		IF NOT DilSendCmd.bBusy THEN
			IF DilSendCmd.bError THEN
				bError := TRUE;
				nErrorId := DilSendCmd.nErrorId;
				bBusy:= FALSE;
			ELSE
				nState := 4;
			END_IF
			DilSendCmd(bExecute:= FALSE);
		ELSE
			RETURN;
		END_IF
	ELSIF nState = 4 THEN	//Ausgangsposition DilSrc erreicht?
		fbGetPlungerPos(bExecute:= TRUE, DilSendCmd:= DilSendCmd, pDilRef:= pDilRefSrc);
		IF NOT fbGetPlungerPos.bBusy THEN
			IF fbGetPlungerPos.bError THEN
				bBusy := FALSE;
				bError := TRUE;
				nErrorId := fbGetPlungerPos.nErrorId;
			ELSE
				nCurPlungerPosSrc := fbGetPlungerPos.nValue;
				IF fbGetPlungerPos.bStatus THEN
					IF nCurPlungerPosSrc = nStartPosSrc THEN
						nState := 5;
					ELSE
						bBusy := FALSE;
						bError := TRUE;
						nErrorId := 333;
					END_IF
				END_IF
			END_IF
			fbGetPlungerPos(bExecute:= FALSE, DilSendCmd:= DilSendCmd);
		ELSE
			RETURN;
		END_IF
	ELSIF nState = 5 THEN	//Ausgangsposition DilDest erreicht?
		fbGetPlungerPos(bExecute:= TRUE, DilSendCmd:= DilSendCmd, pDilRef:= pDilRefDest);
		IF NOT fbGetPlungerPos.bBusy THEN
			IF fbGetPlungerPos.bError THEN
				bBusy := FALSE;
				bError := TRUE;
				nErrorId := fbGetPlungerPos.nErrorId;
			ELSE
				nCurPlungerPosDest := fbGetPlungerPos.nValue;
				IF fbGetPlungerPos.bStatus THEN
					IF nCurPlungerPosDest = nStartPosDest THEN
						IF nPreSteps > 0 THEN
							//DilSrc mit PreSteps Pumpen
							nState := 6;
						ELSIF nPreSteps = 0 THEN
							nState := 8;
						ELSE // < 0
							//DilDest mit PreSteps Pumpen
							nState := 7;
						END_IF
					ELSE
						bBusy := FALSE;
						bError := TRUE;
						nErrorId := 333;
					END_IF
				END_IF
			END_IF
			fbGetPlungerPos(bExecute:= FALSE, DilSendCmd:= DilSendCmd);
		ELSE
			RETURN;
		END_IF
	ELSIF nState = 6 THEN	//DilSrc mit PreSteps pumpen
		fbMoveToPos(nTopSpeed:= DINT_TO_UINT(nSpeedPump), nPosition:= INT_TO_UINT(24000 - nPreSteps), nValvePos:= nValveOutputSrc, bExecute:= TRUE,
					DilSendCmd:= DilSendCmd, pDilRef:= pDilRefSrc);
		IF NOT fbMoveToPos.bBusy THEN
			IF fbMoveToPos.bError THEN
				bBusy := FALSE;
				bError := TRUE;
				nErrorId := fbMoveToPos.nErrorId;
			ELSE
				nCurPlungerPosSrc := pDilRefSrc^.nActPlungerPos;
			END_IF
			fbMoveToPos(bExecute:= FALSE, DilSendCmd:= DilSendCmd, pDilRef:= pDilRefSrc);
			nState := 8;
		ELSE
			RETURN;
		END_IF
	ELSIF nState = 7 THEN	//DilDest mit PreSteps pumpen
		fbMoveToPos(nTopSpeed:= DINT_TO_UINT(nSpeedPump), nPosition:= INT_TO_UINT(-nPreSteps), nValvePos:= nValveOutputDest, bExecute:= TRUE,
					DilSendCmd:= DilSendCmd, pDilRef:= pDilRefDest);
		IF NOT fbMoveToPos.bBusy THEN
			IF fbMoveToPos.bError THEN
				bBusy := FALSE;
				bError := TRUE;
				nErrorId := fbMoveToPos.nErrorId;
			ELSE
				nCurPlungerPosDest := pDilRefDest^.nActPlungerPos;
			END_IF
			fbMoveToPos(bExecute:= FALSE, DilSendCmd:= DilSendCmd, pDilRef:= pDilRefDest);
			nState := 8;
		ELSE
			RETURN;
		END_IF
	ELSIF nState = 8 THEN
		//PumpString DilSrc ermitteln
		//Die beiden Valve-Position (Pump und Reload ermitteln)
		//Damit jeweils der kürzeste Umschaltweg ermittelt wird, werden sie sich gegenseitig als OldPos eingesetzt
		sValvePos := F_GetValveCode(nValveOutputSrc,nValveInputSrc,pDilRefSrc^.eValveType);
		sValvePos2 := F_GetValveCode(nValveInputSrc,nValveOutputSrc,pDilRefSrc^.eValveType);
		IF sValvePos = '' OR sValvePos2 = '' THEN
			bError := FALSE;
			nErrorId := E_ErrorIdDiluter.ERRORID_InvalidValveParam;
			bBusy := FALSE;
			RETURN;
		END_IF
		
		//Muss DilSrc die PastSteps ausführen?
		IF nPostSteps < 0 THEN
			nTotalSteps := nTransferSteps + INT_TO_UINT(-nPostSteps);
		ELSE
			nTotalSteps := nTransferSteps;
		END_IF
		
		sString := F_GetPumpString(nChannel:= pDilRefSrc^.nChannel ,eMode := E_DilPumpMode.MODE_Press, sValvePump:= sValvePos, 
									sValveReload:= sValvePos2, nSpeedPump:= nSpeedPump, nSpeedReload:= nSpeedReload, nTotalSteps:= nTotalSteps,
									nCurPlungerPos:= pDilRefSrc^.nActPlungerPos,bEndless:= FALSE, bFirstReload := FALSE);
		nState := 9;
	END_IF
	
	IF nState = 9 THEN //PumpString DilSrc senden (ohne Execute) + PumpString DilDest ermitteln 
		DilSendCmd(bExecute:= TRUE, bExpectReply:= TRUE, sSendData:= sString);
		IF NOT DilSendCmd.bBusy THEN
			IF DilSendCmd.bError THEN
				bError := TRUE;
				nErrorId := DilSendCmd.nErrorId;
				bBusy:= FALSE;
			ELSE
				//PumpString DilDest ermitteln
				sValvePos := F_GetValveCode(nValveOutputDest,nValveWasteDest,pDilRefDest^.eValveType);
				sValvePos2 := F_GetValveCode(nValveWasteDest,nValveOutputDest,pDilRefDest^.eValveType);
				IF sValvePos = '' OR sValvePos2 = '' THEN
					bError := FALSE;
					nErrorId := E_ErrorIdDiluter.ERRORID_InvalidValveParam;
					bBusy := FALSE;
					RETURN;
				END_IF
				
				//Muss DilSrc die PastSteps ausführen?
				IF nPostSteps > 0 THEN
					nTotalSteps := nTransferSteps + INT_TO_UINT(nPostSteps);
				ELSE
					nTotalSteps := nTransferSteps;
				END_IF
				
				sString := F_GetPumpString(nChannel:= pDilRefDest^.nChannel ,eMode := E_DilPumpMode.MODE_Suck, sValvePump:= sValvePos,
											sValveReload:= sValvePos2, nSpeedPump:= nSpeedPump, nSpeedReload:= nSpeedReload, nTotalSteps:= nTotalSteps,
											nCurPlungerPos:= nCurPlungerPosDest, bEndless:= FALSE, bFirstReload:= FALSE);
				nState := 10;
			END_IF
			DilSendCmd(bExecute:= FALSE);
		ELSE
			RETURN;
		END_IF;
	END_IF

	IF nState = 10 THEN //PumpString DilDest senden (ohne Execute)
		DilSendCmd(bExecute:= TRUE, bExpectReply:= TRUE, sSendData:= sString);
		IF NOT DilSendCmd.bBusy THEN
			IF DilSendCmd.bError THEN
				bError := TRUE;
				nErrorId := DilSendCmd.nErrorId;
				bBusy:= FALSE;
			ELSE
				nState := 11;
				//ChannelCode für TwinDiluter ermitteln und Execute anhängen
				sString := CONCAT(F_GetChannelCodeTwin(pDilRefSrc^.nChannel,pDilRefDest^.nChannel),'R');
			END_IF
			DilSendCmd(bExecute:= FALSE);
		ELSE
			RETURN;
		END_IF;
	END_IF
	
	IF nState = 11 THEN //Execute 'R' an beide Diluter senden
		DilSendCmd(bExecute:= TRUE, bExpectReply:= FALSE, sSendData:= sString);
		IF NOT DilSendCmd.bBusy THEN
			IF DilSendCmd.bError THEN
				bError := TRUE;
				nErrorId := DilSendCmd.nErrorId;
				bBusy:= FALSE;
			ELSE
				nState := 12;
			END_IF
			DilSendCmd(bExecute:= FALSE);
		ELSE
			RETURN;
		END_IF;
	END_IF
	
	IF nState = 12 THEN //DilSrc fertig? (PlungerPos abfragen)
		fbGetPlungerPos(DilSendCmd:= DilSendCmd, pDilRef:= pDilRefSrc, bExecute:= TRUE);
		IF NOT fbGetPlungerPos.bBusy THEN
			IF fbGetPlungerPos.bError THEN
				bError := TRUE;
				nErrorId := fbGetPlungerPos.nErrorId;
				bBusy := FALSE;
			ELSE
				IF fbGetPlungerPos.bStatus THEN
					nState := 13;	
				END_IF
			END_IF
			fbGetPlungerPos(DilSendCmd:= DilSendCmd, bExecute:= FALSE);
		ELSE
			RETURN;
		END_IF
	END_IF
		
	IF nState = 13 THEN //DilDest fertig? (PlungerPos abfragen)
		fbGetPlungerPos(DilSendCmd:= DilSendCmd, pDilRef:= pDilRefDest, bExecute:= TRUE);
		IF NOT fbGetPlungerPos.bBusy THEN
			IF fbGetPlungerPos.bError THEN
				bError := TRUE;
				nErrorId := fbGetPlungerPos.nErrorId;
				bBusy := FALSE;
			ELSE
				IF fbGetPlungerPos.bStatus THEN
					nState := 14;	
				END_IF
			END_IF
			fbGetPlungerPos(DilSendCmd:= DilSendCmd, bExecute:= FALSE);
		ELSE
			RETURN;
		END_IF	
	END_IF
		
	IF nState = 14 THEN //ValvePos DilSrc abfragen
		fbGetValvePos(bExecute:= TRUE, DilSendCmd:= DilSendCmd,	pDilRef:= pDilRefSrc);
		IF NOT fbGetValvePos.bBusy THEN
			IF fbGetValvePos.bError THEN
				bError := TRUE;
				nErrorId := fbGetPlungerPos.nErrorId;
				bBusy := FALSE;
			ELSE
				nState := 15;
			END_IF
			fbGetValvePos(bExecute:= FALSE, DilSendCmd:= DilSendCmd);
		END_IF
	END_IF
		
	IF nState = 15 THEN //ValvePos DilDest abfragen
		fbGetValvePos(bExecute:= TRUE, DilSendCmd:= DilSendCmd,	pDilRef:= pDilRefDest);
		IF NOT fbGetValvePos.bBusy THEN
			IF fbGetValvePos.bError THEN
				bError := TRUE;
				nErrorId := fbGetPlungerPos.nErrorId;
			END_IF
			bBusy := FALSE;
			fbGetValvePos(bExecute:= FALSE, DilSendCmd:= DilSendCmd);
		END_IF
	END_IF
	
ELSE
	IF bBusy THEN
		IF fbGetPlungerPos.bBusy THEN	//FB noch zu Ende führen
			fbGetPlungerPos(bExecute:= TRUE, DilSendCmd:= DilSendCmd);
			IF NOT fbGetPlungerPos.bBusy THEN
				IF fbGetPlungerPos.bError THEN
					bError := TRUE;
					nErrorId := fbGetPlungerPos.nErrorId;
				END_IF
				fbGetPlungerPos(bExecute:= FALSE, DilSendCmd:= DilSendCmd);
				bBusy := FALSE;
				nState := 0;
			END_IF
		ELSIF fbGetValvePos.bBusy THEN	//FB noch zu Ende führen
			fbGetValvePos(bExecute:= TRUE, DilSendCmd:= DilSendCmd);
			IF NOT fbGetValvePos.bBusy THEN
				IF fbGetValvePos.bError THEN
					bError := TRUE;
					nErrorId := fbGetValvePos.nErrorId;
				END_IF
				fbGetValvePos(bExecute:= FALSE, DilSendCmd:= DilSendCmd);
				bBusy := FALSE;
				nState := 0;
			END_IF
		ELSIF fbMoveToPos.bBusy THEN //FB beenden
			fbMoveToPos(bExecute:= FALSE, DilSendCmd:= DilSendCmd);
			IF NOT fbMoveToPos.bBusy THEN
				IF fbMoveToPos.bError THEN
					bError := TRUE;
					nErrorId := fbMoveToPos.nErrorId;
				END_IF
				fbMoveToPos(bExecute:= FALSE, DilSendCmd:= DilSendCmd);
				bBusy := FALSE;
				nState := 0;
			END_IF
		ELSIF DilSendCmd.bBusy THEN	//FB noch zu Ende führen
			DilSendCmd();
			IF NOT DilSendCmd.bBusy THEN
				IF DilSendCmd.bError THEN
					bError := TRUE;
					nErrorId := DilSendCmd.nErrorId;
				END_IF
				DilSendCmd(bExecute:= FALSE);
				bBusy := FALSE;
				nState := 0;
			END_IF
		ELSE
			bBusy := FALSE;
			nState := 0;
		END_IF
	ELSE
		nState := 0;
		bBusy := FALSE;
		bError := FALSE;
		nErrorId := 0;		
	END_IF
END_IF

END_FUNCTION_BLOCK

// ---- Hardware/Diluter/FB_Dil_MoveToPos.TcPOU
FUNCTION_BLOCK FB_Dil_MoveToPos
VAR_INPUT
	bExecute	: BOOL;
	pDilRef		: POINTER TO FB_HwRefDiluter;
	nTopSpeed	: UINT;
	nPosition	: UINT;
	nValvePos	: SINT;	
	
END_VAR
VAR_OUTPUT
	bBusy		: BOOL;
	bError		: BOOL;
	nErrorId	: ERRORID;
END_VAR
VAR
	rTrig : R_TRIG;
	//pDilRefIntern : POINTER TO ST_DiluterRef;
	pDilRefIntern : POINTER TO FB_HwRefDiluter;	
	nState		: USINT;
	sValvePos	: STRING[2];
	sString		: STRING;
	bStatus		: BOOL;	
END_VAR
VAR_IN_OUT
	DilSendCmd 	: FB_Dil_SendCmd;
END_VAR

rTrig(CLK:= bExecute);
IF rTrig.Q THEN
	IF pDilRef = 0 THEN
		bError := TRUE;
		RETURN;	
	ELSE
		pDilRefIntern := pDilRef;
	END_IF	
END_IF

IF bExecute THEN
	IF nState = 0 THEN	//Command senden
		sValvePos := F_GetValveCode(nValvePos,pDilRefIntern^.nActValvePos,pDilRefIntern^.eValveType);
		IF sValvePos = '' THEN
			bError := TRUE;
			nErrorId := E_ErrorIdDiluter.ERRORID_InvalidValveParam;
			RETURN;
		END_IF
		
		sString := CONCAT(USINT_TO_STRING(pDilRefIntern^.nChannel),'v100c100V');	//Startspeed,CutOffSpeed + Kennung für Topspeed
		sString := CONCAT(sString,UINT_TO_STRING(nTopSpeed));	//Topspeed
		sString := CONCAT(sString,sValvePos);					//Ventilposition
		sString := CONCAT(sString,'A');							//Kennung für Move
		sString := CONCAT(sString, UINT_TO_STRING(nPosition));	//Position
		sString := CONCAT(sString,'R');							//Execute-Zeichen	
	
		pDilRefIntern^.bBusy := bBusy := TRUE;
		
		DilSendCmd(bExecute:= TRUE, bExpectReply:= TRUE, sSendData:= sString);
		
		IF NOT DilSendCmd.bBusy THEN
			IF DilSendCmd.bError THEN
				pDilRefIntern^.bBusy := bBusy := FALSE;
				bError := TRUE;
				nErrorId := DilSendCmd.nErrorId;
			ELSE
				pDilRefIntern^.nActValvePos := nValvePos;
				nState := 1;
			END_IF
			DilSendCmd(bExecute:= FALSE);
		END_IF
		
	ELSE //Move-Pos fertig? (Durch Abfrage der Plunger-Pos)
		DilSendCmd(bExecute:= TRUE, bExpectReply:= TRUE, sSendData:= CONCAT(USINT_TO_STRING(pDilRefIntern^.nChannel),'?0'));
		IF NOT DilSendCmd.bBusy THEN
			IF DilSendCmd.bError THEN
				pDilRefIntern^.bBusy := bBusy := FALSE;
				bError := TRUE;
				nErrorId := DilSendCmd.nErrorId;
			ELSE
				IF DilSendCmd.bDataIsNumeric THEN
					pDilRefIntern^.nActPlungerPos := STRING_TO_UINT(DilSendCmd.sReceiveData);
				END_IF
				IF DilSendCmd.bStatus THEN
					pDilRefIntern^.bBusy := bBusy := FALSE;
				END_IF
			END_IF
			DilSendCmd(bExecute:= FALSE);
		END_IF
	END_IF
ELSE
	IF bBusy THEN //DilSendCmd moch zu Ende führen
		DilSendCmd();
		IF NOT DilSendCmd.bBusy THEN
			IF DilSendCmd.bError THEN
				bError := TRUE;
				nErrorId := DilSendCmd.nErrorId;
			END_IF
			DilSendCmd(bExecute:= FALSE);
			pDilRefIntern^.bBusy := bBusy := FALSE;
			nState := 0;
		END_IF
	ELSE
		nState := 0;
		bError := FALSE;
		nErrorId := 0;		
		IF pDilRefIntern > 0 THEN
			pDilRefIntern^.bBusy := bBusy := FALSE;	
		END_IF
	END_IF
END_IF

END_FUNCTION_BLOCK

// ---- Hardware/Diluter/F_GetValveCode.TcPOU
FUNCTION F_GetValveCode : STRING[2]
VAR_INPUT
	nNewValvePos : SINT;
	nOldValvePos : SINT;
	eValveType   : E_DilValveType;
END_VAR
VAR
	bDirRight	: BOOL;	//ValveMovement CW
END_VAR

IF eValveType = E_DilValveType.VALVETYPE_3Way THEN
	//Beim 3-Way-Valve ist keine Drehrichtung zu beachten
	IF nNewValvePos = 1 THEN //Input
		F_GetValveCode := 'I';
	ELSIF nNewValvePos = 2 THEN //Output
		F_GetValveCode := 'O';
	ELSIF nNewValvePos = 3 THEN //Bypass
		F_GetValveCode := 'B';
	END_IF	
ELSIF eValveType = E_DilValveType.VALVETYPE_4Distribution THEN
	//Beim 4-Port-Distribution-Valve wird nach dem kürzestem Weg gesucht ausgehend von "nOldValvePos"
	IF nNewValvePos >= 1 AND nNewValvePos <= 4 THEN
		IF nNewValvePos > nOldValvePos THEN
			bDirRight := TRUE;
		END_IF
		IF ABS(nNewValvePos - nOldValvePos) > 2 THEN
			bDirRight := NOT bDirRight;
		END_IF
		IF bDirRight THEN
			F_GetValveCode := CONCAT('I',SINT_TO_STRING(nNewValvePos));
		ELSE
			F_GetValveCode := CONCAT('O',SINT_TO_STRING(nNewValvePos));
		END_IF		
	END_IF
END_IF

END_FUNCTION

// ---- Hardware/Diluter/F_GetPumpString.TcPOU
FUNCTION F_GetPumpString : STRING[100]
VAR_INPUT
	nChannel		: USINT;
	eMode			: E_DilPumpMode;
	sValvePump		: STRING[2];	//Ventilstellung Pumpen
	sValveReload	: STRING[2];	//Ventilstellung Nachladen
	nSpeedPump		: DINT;		//Gechwindigkeit Pumpen in Halbsteps/s
	nSpeedReload	: DINT;		//Gechwindigkeit Nachladen in Halbsteps/s
	nTotalSteps		: UDINT;	//Gesamtanzahl in Microsteps
	nCurPlungerPos	: UINT;		
	bEndless		: BOOL;		//Die Microsteps werden ignortiert und es wird endloss gepumpt
	bFirstReload	: BOOL;		//Es wird immer erst in die Ausgangsposition gefahren, damit am Anfang kein Teilhub entsteht.
END_VAR
VAR
	nPosition		: UDINT;		//zwischengespeicherte Position
	nFullStrokes	: UDINT;		//ganze Hübe
	nFirstPartSteps	: UDINT;		//Steps erster Teilhub
	nLastPartSteps	: UDINT;		//Steps letzter Teilhub
	sString			: STRING[100];	//Sendestring
	sTopSpeedPump		: STRING(7);//Topspeed als String
	sTopSpeedReload		: STRING(7);//Topspeed als String
	sFirstPartStepsP	: STRING(7);//FirstPartSteps als String mit Bezeichner P (relative Positionierung Saugen)
	sFirstPartStepsD	: STRING(7);//FirstPartSteps als String mit Bezeichner D (relative Positionierung Pumpen)
	sLastPartStepsP		: STRING(7);//FirstPartSteps als String mit Bezeichner P (relative Positionierung Saugen)
	sLastPartStepsD		: STRING(7);//FirstPartSteps als String mit Bezeichner D (relative Positionierung Pumpen)
	sFullStrokes		: STRING(5);//volle Hübe als String mit Bezeichner G (Schleifenende)	
END_VAR

VAR_OUTPUT
	nPlungerMoves	: UINT;
END_VAR

IF bFirstReload THEN
	//in diesem Fall muss die aktuelle Plungerpos überschrieben werden auf den Wert der ReloadPos
	IF eMode = E_DilPumpMode.MODE_Suck THEN
		IF nCurPlungerPos = 0 THEN //Fahrt zu ReloadPos nicht notwendig.
			bFirstReload := FALSE;
		ELSE
			nCurPlungerPos := 0;
		END_IF
	ELSE
		IF nCurPlungerPos = 24000 THEN //Fahrt zu ReloadPos nicht notwendig.
			bFirstReload := FALSE;
		ELSE
			nCurPlungerPos := 24000;	
		END_IF
	END_IF
END_IF

//Bezugsposition errechnen
IF eMode = E_DilPumpMode.MODE_Suck THEN	//Saugen
	nPosition := UINT_TO_UDINT(24000 - nCurPlungerPos);
ELSIF eMode = E_DilPumpMode.MODE_Press THEN	//Pumpen
	nPosition := UINT_TO_UDINT(nCurPlungerPos);
END_IF

//Hübe und Teilhübe berechnen
IF nCurPlungerPos > 0 AND nCurPlungerPos < 24000 THEN	//Kolben ist weder oben noch unten
	IF bEndless THEN
		nFirstPartSteps := nPosition;
	ELSIF nTotalSteps <= nPosition THEN
		nFirstPartSteps := nTotalSteps;
		nFullStrokes := 0;
		nLastPartSteps := 0; 
	ELSE
		nFirstPartSteps := nPosition;
		nLastPartSteps := (nTotalSteps - nFirstPartSteps) MOD 24000;
		nFullStrokes := (nTotalSteps - nLastPartSteps) / 24000;
	END_IF
ELSE	//Kolben ist oben oder unten
	IF NOT bEndless THEN
		IF nTotalSteps < 24000 THEN
			nFirstPartSteps := nTotalSteps;
			nFullStrokes := 0;
			nLastPartSteps := 0; 
		ELSE
			nFirstPartSteps := 0;
			nLastPartSteps := nTotalSteps MOD 24000;
			nFullStrokes := (nTotalSteps - nLastPartSteps) / 24000; 
		END_IF		
	END_IF	
END_IF

//Teilstrings vorbereiten
sString := CONCAT(USINT_TO_STRING(nChannel),'v400');				//Diluternummer, Startgeschwindigkeit
sTopSpeedPump := CONCAT('V', DINT_TO_STRING(nSpeedPump));			//TopSpeed Pumpen in in String mit Bezeichner umwandeln
sTopSpeedReload := CONCAT('V', DINT_TO_STRING(nSpeedReload));			//TopSpeed Nachladen in in String mit Bezeichner umwandeln
sFirstPartStepsP := CONCAT('P', UDINT_TO_STRING(nFirstPartSteps));	//FirstPartSteps in String mit Bezeichner umwandeln
sFirstPartStepsD := CONCAT('D', UDINT_TO_STRING(nFirstPartSteps));	//FirstPartSteps in String mit Bezeichner umwandeln
sLastPartStepsP := CONCAT('P', UDINT_TO_STRING(nLastPartSteps));		//LastPartSteps in String mit Bezeichner umwandeln
sLastPartStepsD := CONCAT('D', UDINT_TO_STRING(nLastPartSteps));		//LastPartSteps in String mit Bezeichner umwandeln
sFullStrokes := CONCAT('G', UDINT_TO_STRING(nFullStrokes));			//FullStrokes in String mit Bezeichner umwandeln			
nPosition := UINT_TO_UDINT(nCurPlungerPos);
//############## M O D E :  S A U G E N ##############################################################################################
IF eMode = E_DilPumpMode.MODE_Suck THEN	//Saugen
	
	IF bFirstReload THEN //in ReloadPos (oben) fahren
		sString := CONCAT(sString, sTopSpeedReload);	//Topspeed >Nachladen<
		sString := CONCAT(sString, sValveReload);		//Ventilstellung >Nachladen<
		sString := CONCAT(sString, 'A0');
	END_IF
	
	IF nFirstPartSteps > 0 THEN
		//Wenn Position = 24000 dann um nFirstPartSteps nach oben fahren
		IF nPosition = 24000 THEN	//Nachladen
			sString := CONCAT(sString, sTopSpeedReload);	//Topspeed >Nachladen<
			sString := CONCAT(sString, sValveReload);		//Ventilstellung >Nachladen<
			sString := CONCAT(sString, sFirstPartStepsD);	//Move nach oben um >nLastFirstSteps<
			nPosition := 24000 - nFirstPartSteps;
			nPlungerMoves := nPlungerMoves + 1;						
		END_IF
		//um nFirstPartSteps nach unten fahren
		sString := CONCAT(sString, sTopSpeedPump);		//Topspeed >Pumpen<
		sString := CONCAT(sString, sValvePump);			//Ventilstellung >Pumpen<
		sString := CONCAT(sString, sFirstPartStepsP);	//FirstPartSteps
		nPlungerMoves := nPlungerMoves + 1;
		//Neue imaginäre Position setzen
		nPosition := nPosition + nFirstPartSteps;
	END_IF
	
	IF nFullStrokes > 0 OR bEndless THEN
		//Wenn Position = 24000 dann nach Top fahren
		IF nPosition = 24000 THEN
			sString := CONCAT(sString, sTopSpeedReload);	//Topspeed >Nachladen<
			sString := CONCAT(sString, sValveReload);		//Ventilstellung >Nachladen<
			sString := CONCAT(sString, 'A0');	//Move nach TOP
			nPlungerMoves := nPlungerMoves + 1;
			nPosition := 0;
		END_IF
		//1* Saugen
		sString := CONCAT(sString, sTopSpeedPump);		//Topspeed >Pumpen<
		sString := CONCAT(sString, sValvePump);			//Ventilstellung >Pumpen<
		sString := CONCAT(sString, 'A24000');		//Move nach >Unten<
		nPlungerMoves := nPlungerMoves + UDINT_TO_UINT(nFullStrokes);
		//Wenn nFullStrokes > 1 dann Schleife mit Nachladen/Saugen
		IF nFullStrokes > 1 OR bEndless THEN
			sString := CONCAT(sString,'g');									//Schleifenkopf
			//Nachladen
			sString := CONCAT(sString, sTopSpeedReload);					//Topspeed >Nachladen<
			sString := CONCAT(sString, sValveReload);						//Ventilstellung >Nachladen<
			sString := CONCAT(sString, 'A0');								//Move nach >Oben<
			//Saugen
			sString := CONCAT(sString, sTopSpeedPump);						//Topspeed >Pumpen<
			sString := CONCAT(sString, sValvePump);							//Ventilstellung >Pumpen<
			sString := CONCAT(sString, 'A24000');							//Move nach >Unten<
			sString := CONCAT(sString,'G');									//Schleifenfuß Bezeichner
			IF bEndless THEN
				sString := CONCAT(sString,'0');								//Schleifenfuss - unendliche Anzahl Durchläufe
			ELSE
				sString := CONCAT(sString,UDINT_TO_STRING(nFullStrokes -1));//Schleifenfuss - Anzahle Durchläufe minus 1
			END_IF
			
		END_IF					
		//neue imaginäre Position setzen
		nPosition := 24000;
	END_IF
	
	IF nLastPartSteps > 0 THEN
		//Wenn Position = 24000 dann um nLastPartSteps nach oben fahren
		IF nPosition = 24000 THEN
			sString := CONCAT(sString, sTopSpeedReload);		//Topspeed >Nachladen<
			sString := CONCAT(sString, sValveReload);			//Ventilstellung >Nachladen<
			sString := CONCAT(sString,sLastPartStepsD);			//Move nach oben um >nLastFirstSteps<
		END_IF
		//Saugen
		sString := CONCAT(sString, sTopSpeedPump);				//Topspeed Pumpen
		sString := CONCAT(sString, sValvePump);					//Ventilstellung "Pumpen"
		sString := CONCAT(sString, sLastPartStepsP);			//FirstPartSteps
		//um  nLastPartSteps nach unten fahren	
	END_IF
	
	
//############## M O D E :  P U M P E N ##############################################################################################			
ELSIF eMode = E_DilPumpMode.MODE_Press THEN	//Pumpen
	
	IF bFirstReload THEN //in ReloadPos (unten) fahren
		sString := CONCAT(sString, sTopSpeedReload);	//Topspeed >Nachladen<
		sString := CONCAT(sString, sValveReload);		//Ventilstellung >Nachladen<
		sString := CONCAT(sString, 'A24000');
	END_IF
	
	IF nFirstPartSteps > 0 THEN
		//Wenn Position = 0 dann um nFirstPartSteps nach unten fahren
		IF nPosition = 0 THEN
			sString := CONCAT(sString, sTopSpeedReload);	//Topspeed >Nachladen<
			sString := CONCAT(sString, sValveReload);		//Ventilstellung >Nachladen<
			sString := CONCAT(sString,sFirstPartStepsP);	//Move nach unten um >nLastFirstSteps<
			nPosition := nFirstPartSteps;						
		END_IF
		//um nFirstPartSteps nach oben fahren
		sString := CONCAT(sString, sTopSpeedPump);		//Topspeed >Pumpen<
		sString := CONCAT(sString, sValvePump);			//Ventilstellung >Pumpen<
		sString := CONCAT(sString, sFirstPartStepsD);	//FirstPartSteps
		//Neue imaginäre Position setzen
		nPosition := nPosition - nFirstPartSteps;
	END_IF
	
	IF nFullStrokes > 0 OR bEndless THEN
		//Wenn Position = 0 dann nach Bottom fahren
		IF nPosition = 0 THEN
			sString := CONCAT(sString, sTopSpeedReload);	//Topspeed >Nachladen<
			sString := CONCAT(sString, sValveReload);		//Ventilstellung >Nachladen<
			sString := CONCAT(sString, 'A24000');			//Move nach Bottom
			nPosition := 24000;
		END_IF
		//1* Pumpen
		sString := CONCAT(sString, sTopSpeedPump);			//Topspeed >Pumpen<
		sString := CONCAT(sString, sValvePump);				//Ventilstellung >Pumpen<
		sString := CONCAT(sString, 'A0');					//Move nach >Oben<
		//Wenn nFullStrokes > 1 dann Schleife mit Nachladen/Saugen
		IF nFullStrokes > 1 OR bEndless THEN
			sString := CONCAT(sString,'g');									//Schleifenkopf
			//Nachladen
			sString := CONCAT(sString, sTopSpeedReload);					//Topspeed >Nachladen<
			sString := CONCAT(sString, sValveReload);						//Ventilstellung >Nachladen<
			sString := CONCAT(sString, 'A24000');							//Move nach >Unten<
			//Saugen
			sString := CONCAT(sString, sTopSpeedPump);						//Topspeed >Pumpen<
			sString := CONCAT(sString, sValvePump);							//Ventilstellung >Pumpen<
			sString := CONCAT(sString, 'A0');								//Move nach >Oben<
			sString := CONCAT(sString,'G');									//Schleifenfuß Bezeichner
			IF bEndless THEN
				sString := CONCAT(sString,'0');								//Schleifenfuss - unendliche Anzahl Durchläufe
			ELSE
				sString := CONCAT(sString,UDINT_TO_STRING(nFullStrokes -1));//Schleifenfuss - Anzahle Durchläufe minus 1	
			END_IF
			
		END_IF					
		//neue imaginäre Position setzen
		nPosition := 0;
	END_IF
	
	IF nLastPartSteps > 0 THEN
		//Wenn Position = 0 dann um nLastPartSteps nach unten fahren
		IF nPosition = 0 THEN
			sString := CONCAT(sString, sTopSpeedReload);		//Topspeed >Nachladen<
			sString := CONCAT(sString, sValveReload);			//Ventilstellung >Nachladen<
			sString := CONCAT(sString,sLastPartStepsP);			//Move nach unten um >nLastFirstSteps<
		END_IF
		//Pumpen
		sString := CONCAT(sString, sTopSpeedPump);				//Topspeed >Pumpen<
		sString := CONCAT(sString, sValvePump);					//Ventilstellung >Pumpen<
		sString := CONCAT(sString, sLastPartStepsD);			//FirstPartSteps
	END_IF
END_IF

F_GetPumpString := sString;

END_FUNCTION

// ---- Hardware/Diluter/F_GetChannelCodeTwin.TcPOU
FUNCTION F_GetChannelCodeTwin : STRING[1]
VAR_INPUT
	nChannel1 : USINT;
	nChannel2 : USINT;
END_VAR
VAR
END_VAR

IF nChannel1 = 1 AND nChannel2 = 2 OR nChannel1 = 2 AND nChannel2 = 1 THEN
	F_GetChannelCodeTwin := 'A';
ELSIF nChannel1 = 3 AND nChannel2 = 4 OR nChannel1 = 4 AND nChannel2 = 3 THEN
	F_GetChannelCodeTwin := 'C';
ELSIF nChannel1 = 5 AND nChannel2 = 6 OR nChannel1 = 6 AND nChannel2 = 5 THEN
	F_GetChannelCodeTwin := 'E';
ELSIF nChannel1 = 7 AND nChannel2 = 8 OR nChannel1 = 8 AND nChannel2 = 7 THEN
	F_GetChannelCodeTwin := 'G';
ELSIF nChannel1 = 9 AND nChannel2 = 10 OR nChannel1 = 10 AND nChannel2 = 9 THEN
	F_GetChannelCodeTwin := 'I';
ELSIF nChannel1 = 11 AND nChannel2 = 12 OR nChannel1 = 12 AND nChannel2 = 11 THEN
	F_GetChannelCodeTwin := 'K';
ELSIF nChannel1 = 13 AND nChannel2 = 14 OR nChannel1 = 14 AND nChannel2 = 13 THEN
	F_GetChannelCodeTwin := 'M';
ELSE //Andere Paarkombinationen gibt es nicht, da Diluter immer direkt nebeneinander liegen müssen.
	F_GetChannelCodeTwin := '_'; //Das ist der Code für alle Diluter
	
END_IF

END_FUNCTION

// ---- Hardware/Diluter/FB_Dil_MoveValve.TcPOU
FUNCTION_BLOCK FB_Dil_MoveValve
VAR_INPUT
	bExecute	: BOOL;
	nValvePos	: SINT;
END_VAR
VAR_OUTPUT
	bBusy		: BOOL;
	bError		: BOOL;
	nErrorId	: ERRORID;
	
END_VAR
VAR
	nState		: USINT;
	sValvePos	: STRING[2];
	sString		: STRING;
	bStatus		: BOOL;
	nCurrentPos	: SINT;
END_VAR
VAR_IN_OUT
	pDilRef		: POINTER TO FB_HwRefDiluter;
	DilSendCmd 	: FB_Dil_SendCmd;
END_VAR

IF pDilRef = 0 THEN
	bError := TRUE;
	RETURN;
END_IF

IF bExecute THEN
	IF nState = 0 THEN	//Command senden
		sValvePos := F_GetValveCode(nValvePos,pDilRef^.nActValvePos,pDilRef^.eValveType);
		IF sValvePos = '' THEN
			bError := TRUE;
			nErrorId := E_ErrorIdDiluter.ERRORID_InvalidValveParam;
			RETURN;
		END_IF
		sString := CONCAT(USINT_TO_STRING(pDilRef^.nChannel),sValvePos);	//Ventilposition
		sString := CONCAT(sString,'R');							//Execute-Zeichen		
		bBusy := TRUE;
		DilSendCmd(bExecute:= TRUE, bExpectReply:= TRUE, sSendData:= sString);
		
		IF NOT DilSendCmd.bBusy THEN
			IF DilSendCmd.bError THEN
				bError := TRUE;
				nErrorId := DilSendCmd.nErrorId;
				bBusy := FALSE;
			ELSE
				nState := 1;
			END_IF
			DilSendCmd(bExecute:= FALSE);
		END_IF
	ELSE //MoveValve fertig? (Durch Abfrage der Valve-Pos)
		DilSendCmd(bExecute:= TRUE, bExpectReply:= TRUE, sSendData:= CONCAT(USINT_TO_STRING(pDilRef^.nChannel),'?6'));
		
		IF NOT DilSendCmd.bBusy THEN
			IF DilSendCmd.bError THEN
				bError := TRUE;
				nErrorId := DilSendCmd.nErrorId;
			ELSE
				IF DilSendCmd.bStatus THEN
					IF DilSendCmd.bDataIsNumeric THEN
						nCurrentPos := STRING_TO_SINT(DilSendCmd.sReceiveData);
					ELSE
						sString := F_ToUCase(DilSendCmd.sReceiveData);
						IF sString = 'I' THEN
							nCurrentPos := 1;
						ELSIF sString = 'O' THEN
							nCurrentPos := 2;
						ELSIF sString = 'B' THEN
							nCurrentPos := 3;
						ELSIF sString = 'E' THEN
							nCurrentPos := 4;
						END_IF
					END_IF
					pDilRef^.nActValvePos := nCurrentPos;				
					bBusy := FALSE;
				END_IF
			END_IF
			DilSendCmd(bExecute:= FALSE);
		END_IF
	END_IF
ELSE
	IF bBusy THEN //DilSendCmd moch zu Ende führen
		DilSendCmd();
		IF NOT DilSendCmd.bBusy THEN
			IF DilSendCmd.bError THEN
				bError := TRUE;
				nErrorId := DilSendCmd.nErrorId;
			END_IF
			DilSendCmd(bExecute:= FALSE);
			bBusy := FALSE;
			nState := 0;
		END_IF
	ELSE
		nState := 0;
		bBusy := FALSE;
		bError := FALSE;
		nErrorId := 0;		
	END_IF
END_IF

END_FUNCTION_BLOCK

// ---- Hardware/Diluter/FB_Dil_Pump.TcPOU
FUNCTION_BLOCK FB_Dil_Pump
VAR_INPUT
	eMode			: E_DilPumpMode;
	nValvePosPump	: SINT;		//Ventilstellung Pumpen
	nValvePosReload	: SINT;		//Ventilstellung Nachladen
	nSpeedPump		: DINT;		//Gechwindigkeit Pumpen in Halbsteps/s
	nSpeedReload	: DINT;		//Gechwindigkeit Nachladen in Halbsteps/s
	nTotalSteps		: UDINT;	//Gesamtanzahl in Microsteps
	bEndless		: BOOL;		//Dauerpumpen (nTotalSteps wird ignoriert)
	bFirstReload	: BOOL;		//Es wird zuerst nachgeladen
	bExecute		: BOOL;	
END_VAR
VAR_OUTPUT
	bBusy		: BOOL;
	bError		: BOOL;
	nErrorId	: ERRORID;
END_VAR
VAR
	nState				: USINT;
	bStatus				: BOOL;	
	nFullStrokes		: UDINT;		//ganze Hübe
	nFirstPartSteps		: UDINT;		//Steps erster Teilhub
	nLastPartSteps		: UDINT;		//Steps letzter Teilhub
	nPosition			: UDINT;		//zwischengespeicherte Position
	sString				: STRING[100];	//Sendestring
	sValvePosPump		: STRING[2];
	sValvePosReload		: STRING[2];
	
	fbGetValvePos		: FB_Dil_GetValvePos;
	fbGetPlungerPos		: FB_Dil_GetPlungerPos;
	
	nPlungerMoves		: UINT;
	
	bPlungerNotWithinRange : BOOL;	//tritt manchmal auf, wenn Diluter durch Terminate gestoppt wird
	
END_VAR

VAR_IN_OUT
	DilSendCmd 	: FB_Dil_SendCmd;
	pDilRef		: POINTER TO FB_HwRefDiluter;
END_VAR

IF pDilRef = 0 THEN
	bError := TRUE;
	RETURN;
END_IF

IF bExecute THEN
	IF nState = 0 THEN //aktuelle Position ermitteln
		sValvePosPump := F_GetValveCode(nValvePosPump, nValvePosReload ,pDilRef^.eValveType);
		IF sValvePosPump = '' THEN
			bError := TRUE;
			nErrorId := E_ErrorIdDiluter.ERRORID_InvalidValveParam;
			RETURN;
		END_IF
		sValvePosReload := F_GetValveCode(nValvePosReload, nValvePosPump ,pDilRef^.eValveType);
		IF sValvePosReload = '' THEN
			bError := TRUE;
			nErrorId := E_ErrorIdDiluter.ERRORID_InvalidValveParam;
			RETURN;
		END_IF
	
		bBusy := TRUE;
		fbGetPlungerPos(bExecute:= TRUE, DilSendCmd:= DilSendCmd, pDilRef:= pDilRef);
		IF NOT fbGetPlungerPos.bBusy THEN
			IF fbGetPlungerPos.bError THEN
				bBusy := FALSE;
				bError := TRUE;
				nErrorId := fbGetPlungerPos.nErrorId;
			ELSE
				//PlungerPos steht in "pDilRef"
				//für den Fall, dass Plunger > 24000 ist (kann durch Terminate zu ungünstigem Zeitpunkt enstehen)
				IF pDilRef^.nActPlungerPos < 0 THEN
					bPlungerNotWithinRange := TRUE;
					nState := 2;
					sString := CONCAT(USINT_TO_STRING(pDilRef^.nChannel),'A0R');
				ELSIF pDilRef^.nActPlungerPos > 24000 THEN
					bPlungerNotWithinRange := TRUE;
					sString := CONCAT(USINT_TO_STRING(pDilRef^.nChannel),'A24000R');
					nState := 2;
				ELSE
					nState := 1;	
				END_IF
				
			END_IF
			fbGetPlungerPos(bExecute:= FALSE, DilSendCmd:= DilSendCmd, pDilRef:= pDilRef);
		END_IF
	END_IF
	
	IF nState = 1 THEN //Sende-String berechnen und Execute'R' anhängen
		sValvePosPump := F_GetValveCode(nValvePosPump, nValvePosReload, pDilRef^.eValveType);
		sValvePosReload := F_GetValveCode(nValvePosReload, nValvePosPump, pDilRef^.eValveType);
		sString := CONCAT(F_GetPumpString(nChannel:= pDilRef^.nChannel, eMode:= eMode, sValvePump:= sValvePosPump, 
							sValveReload:= sValvePosReload, nSpeedPump:= nSpeedPump, nSpeedReload:= nSpeedReload, nTotalSteps:= nTotalSteps,
							pDilRef^.nActPlungerPos,nPlungerMoves=>nPlungerMoves, bEndless:= bEndless, bFirstReload:= bFirstReload),'R');
		nState := 2;
	END_IF
	
	IF nState = 2 THEN //String senden
		DilSendCmd(bExecute:= TRUE, bExpectReply:= TRUE, sSendData:= sString);
		IF NOT DilSendCmd.bBusy THEN
			IF DilSendCmd.bError THEN
				bBusy := FALSE;
				bError := TRUE;
				nErrorId := DilSendCmd.nErrorId;
			END_IF
			DilSendCmd(bExecute:= FALSE);
			nState := 3;
		END_IF
	ELSIF nState = 3 THEN //Valve-Pos abfragen bis Status fertig meldet
		fbGetValvePos(pDilRef:= pDilRef, bExecute:= TRUE, DilSendCmd:= DilSendCmd);
		IF NOT fbGetValvePos.bBusy THEN
			IF fbGetValvePos.bError THEN
				bBusy := FALSE;
				bError := TRUE;
				nErrorId := fbGetValvePos.nErrorId;
			ELSE
				IF fbGetValvePos.bStatus THEN
					IF bPlungerNotWithinRange THEN
						bPlungerNotWithinRange := FALSE;
						nState := 0;
					ELSE
						nState := 4;	
					END_IF
				END_IF
			END_IF
			fbGetValvePos(bExecute:= FALSE, DilSendCmd:= DilSendCmd, pDilRef:= pDilRef);
		END_IF
	ELSIF nState = 4 THEN //Plunger-Pos ermitteln
		fbGetPlungerPos(bExecute:= TRUE, DilSendCmd:= DilSendCmd, pDilRef:= pDilRef);
		IF NOT fbGetPlungerPos.bBusy THEN
			IF fbGetPlungerPos.bError THEN
				bError := TRUE;
				nErrorId := fbGetPlungerPos.nErrorId;
			END_IF
			fbGetPlungerPos(bExecute:= FALSE, DilSendCmd:= DilSendCmd, pDilRef:= pDilRef);
			bBusy := FALSE;
		END_IF
	END_IF
ELSE
	IF bBusy THEN
		IF fbGetPlungerPos.bBusy THEN	//FB noch zu Ende führen
			fbGetPlungerPos(bExecute:= TRUE, DilSendCmd:= DilSendCmd, pDilRef:= pDilRef);
			IF NOT fbGetPlungerPos.bBusy THEN
				IF fbGetPlungerPos.bError THEN
					bError := TRUE;
					nErrorId := fbGetPlungerPos.nErrorId;
				END_IF
				fbGetPlungerPos(bExecute:= FALSE, DilSendCmd:= DilSendCmd, pDilRef:= pDilRef);
				bBusy := FALSE;
				nState := 0;
			END_IF
		ELSIF fbGetValvePos.bBusy THEN	//FB noch zu Ende führen
			fbGetValvePos(bExecute:= TRUE,	DilSendCmd:= DilSendCmd, pDilRef:= pDilRef);
			IF NOT fbGetValvePos.bBusy THEN
				IF fbGetValvePos.bError THEN
					bBusy := FALSE;
					bError := TRUE;
					nErrorId := fbGetValvePos.nErrorId;
				END_IF
				fbGetValvePos(bExecute:= FALSE, DilSendCmd:= DilSendCmd, pDilRef:= pDilRef);
				bBusy := FALSE;
				nState := 0;
			END_IF			
		ELSIF DilSendCmd.bBusy THEN	//FB noch zu Ende führen
			DilSendCmd();
			IF NOT DilSendCmd.bBusy THEN
				IF DilSendCmd.bError THEN
					bError := TRUE;
					nErrorId := DilSendCmd.nErrorId;
				END_IF
				DilSendCmd(bExecute:= FALSE);
				bBusy := FALSE;
				nState := 0;
			END_IF
		ELSE
			bBusy := FALSE;
			nState := 0;
		END_IF
	ELSE
		nState := 0;
		bBusy := FALSE;
		bError := FALSE;
		bEndless := FALSE;
		bFirstReload := FALSE;
		nErrorId := 0;		
	END_IF
END_IF

END_FUNCTION_BLOCK

// ---- Hardware/Diluter/FB_Dil_Stop.TcPOU
FUNCTION_BLOCK FB_Dil_Stop
VAR_INPUT
	bExecute	: BOOL;
	pDilRef1	: POINTER TO FB_HwRefDiluter;
	pDilRef2	: POINTER TO FB_HwRefDiluter;
END_VAR
VAR_OUTPUT
	bBusy		: BOOL;
	bError		: BOOL;
	nErrorId	: ERRORID;
END_VAR
VAR
	rTrig 		  : R_TRIG;
	sChannel	: STRING[1];
	bExpectReply : BOOL;
	nChannel1	: USINT;
	nChannel2	: USINT;
END_VAR
VAR_IN_OUT
	DilSendCmd 	: FB_Dil_SendCmd;
END_VAR

rTrig(CLK:= bExecute);
IF rTrig.Q THEN
	IF pDilRef1 = 0 THEN
		bError := TRUE;
		RETURN;	
	ELSE
		nChannel1 := pDilRef1^.nChannel;
		IF pDilRef2 > 0 THEN
			nChannel2 := pDilRef2^.nChannel;
		ELSE
			nChannel2 := 0;
		END_IF
	END_IF
	sChannel := F_GetChannelCodeTwin(nChannel1,nChannel2);
	IF ASC(sChannel) >= 16#31 AND ASC(sChannel) <= 16#39 THEN	//Inhalt numerisch -> genau ein Kanal
		bExpectReply := TRUE; //Antwort vom Diluter wird erwartet
	ELSE
		bExpectReply := FALSE; //keine Antwort vom Diluter möglich
	END_IF
END_IF

IF bExecute THEN
	bBusy := TRUE;
	DilSendCmd(bExecute:= TRUE, bExpectReply:= bExpectReply, sSendData:= CONCAT(sChannel,'T'));
	
	IF NOT DilSendCmd.bBusy THEN
		IF DilSendCmd.bError THEN
			bError := TRUE;
			nErrorId := DilSendCmd.nErrorId;
		END_IF
		DilSendCmd(bExecute:= FALSE);
		bBusy := FALSE;
	END_IF	
ELSE
	DilSendCmd(bExecute:= FALSE);
	bBusy := FALSE;
	bError := FALSE;
	nErrorId := 0;
	pDilRef1 := 0;
	pDilRef2 := 0;
END_IF

END_FUNCTION_BLOCK

// ---- Hardware/Diluter/F_DilFlowToSpeed.TcPOU
FUNCTION F_DilFlowToSpeed : DINT
VAR_INPUT
	nFlow : DINT; //Flow in 10tel µl/sec
	nSyringeSize : DINT; //Spritzengröße in µl
END_VAR
VAR
	rFlow : REAL;
	rSyringe : REAL;
END_VAR

rFlow := DINT_TO_REAL(nFlow);
rSyringe := DINT_TO_REAL(nSyringeSize);
//Speed wird in Halbsteps/sec angegeben -> 1 voller Hub entspricht 6000 Halbsteps
F_DilFlowToSpeed := REAL_TO_DINT(rFlow * 6000.0 / rSyringe / 10.0);

END_FUNCTION

// ---- Hardware/Diluter/F_DilQuantityToMicroSteps.TcPOU
FUNCTION F_DilQuantityToMicroSteps : UDINT
VAR_INPUT
	nQuantity : DINT; //Menge in 10tel µl
	nSyringeSize : DINT; //Spritzengröße in µl
END_VAR
VAR
	rQuantity : REAL;
	rSyringe : REAL;
END_VAR

rQuantity := DINT_TO_REAL(nQuantity);
rSyringe := DINT_TO_REAL(nSyringeSize);
//1 voller HUB (Volumen Spritze) entspricht 24000 Mircosteps
F_DilQuantityToMicroSteps := REAL_TO_UDINT(rQuantity * 24000.0 / rSyringe / 10.0);

END_FUNCTION

// ---- Objects/Devices/FB_Diluter3Inputs.TcPOU
FUNCTION_BLOCK FB_Diluter3Inputs EXTENDS FB_Diluter IMPLEMENTS I_Device

VAR
	aLiquidBottle		: ARRAY[1..3] OF USINT;
 	aValvePosInput 		: ARRAY[1..3] OF SINT;
	nCurrentBottleNr 	: USINT;
	nInput				: USINT;
END_VAR

SUPER^();

ACTION A_Prepare:
stError.POUState := nStateAction;

IF nStateAction = 0 THEN
	nStateAction := 1;
	IF ePrepareMode = E_DilPrepareMode.ForAspirate THEN
		//Abstand von ganz unten zu aktueller Pos muss mind TotalSteps betragen
		nSetPosPlunger := UDINT_TO_UINT(24000 - nTotalSteps);
		//ValvePosition wird bereits in M_ExeAction() gestetzt
		IF nSetPosPlunger >= pDiluterRef1^.nActPlungerPos THEN	//Kolbenposition breits passend
			//weiter zu MoveValve
			nStateAction := 2;
		END_IF
	ELSE //ForDispense
		nSetPosPlunger := UDINT_TO_UINT(nTotalSteps);
		//ValvePosition wird bereits in M_ExeAction() gestetzt
		IF nSetPosPlunger <= pDiluterRef1^.nActPlungerPos THEN	//Kolbenposition bereits passend
			//weiter zu MoveValve
			nStateAction := 2;
		END_IF
	END_IF			
END_IF

IF nStateAction = 1 THEN	//Move plunger
	fbMoveToPos(bExecute:= TRUE, pDilRef:= pDiluterRef1, nTopSpeed:= DINT_TO_UINT(nSpeedReload), 
				nPosition:= nSetPosPlunger, DilSendCmd:= fbSendCmd);
	IF NOT fbMoveToPos.bBusy THEN
		IF fbMoveToPos.bError THEN
			stError.ErrorId := fbMoveToPos.nErrorId;
			nStateAction := 99;
		ELSE
			nStateAction := 2;
		END_IF
		fbMoveToPos(bExecute:= FALSE, pDilRef:= pDiluterRef1, DilSendCmd:= fbSendCmd);
	END_IF
END_IF

IF nStateAction = 2 THEN	//Move valve
	fbMoveValve(bExecute:= TRUE, nValvePos:= nValvePosOutput, pDilRef:= pDiluterRef1, DilSendCmd:= fbSendCmd);
	IF NOT fbMoveValve.bBusy THEN
		IF fbMoveValve.bError THEN
			stError.ErrorId := fbMoveValve.nErrorId;
			nStateAction := 99;
		ELSE
			nStateAction := 80;
		END_IF
		fbMoveValve(bExecute:= FALSE, pDilRef:= pDiluterRef1, DilSendCmd:= fbSendCmd);
	END_IF
END_IF

//Abbrechen
IF nStateAction = 70 THEN
	IF fbMoveToPos.bBusy THEN
		fbMoveToPos(bExecute:= FALSE, DilSendCmd:= fbSendCmd, pDilRef:= pDiluterRef1);
	ELSE
		nStateAction := 71;
	END_IF
END_IF

IF nStateAction = 71 THEN
	fbStop(bExecute:= TRUE, DilSendCmd:= fbSendCmd, pDilRef1 := pDiluterRef1);
	IF NOT fbStop.bBusy THEN
		IF fbStop.bError THEN
			nStateAction := 99;
			stError.ErrorId := fbStop.nErrorId;
		ELSE
			nStateAction := 80;
		END_IF
		fbStop(bExecute:= FALSE, DilSendCmd:= fbSendCmd);
	END_IF	
END_IF
//Ende Abbrechen

//Errorhandling
IF nStateAction = 99 THEN
	stError.Cmd := E_Action.ACTION_DilPrepare;
	stError.POUAction := E_POUACT.POUACT_A_Prepare;
	fbErrorList.M_Add(stError);
END_IF
END_ACTION

ACTION A_Pump:
stError.POUState := nStateAction;

IF nStateAction = 0 THEN
	//BottleStates abfragen
	stError.ErrorId := M_CheckBottles(nCurrentBottleNr);
	IF stError.ErrorId > 0 THEN
		nStateAction := 70;
		nStateNext := 99;
		RETURN;
	END_IF	
	
	nStateNext := 80;
	fbPump(eMode:= ePumpMode, nValvePosPump:= nValvePosPump, nValvePosReload:= nValvePosReload, 
			nSpeedPump:= nSpeedPump, nSpeedReload:= nSpeedReload, nTotalSteps:= nTotalSteps,
			bExecute:= TRUE, DilSendCmd:= fbSendCmd, pDilRef:= pDiluterRef1);
	IF NOT fbPump.bBusy THEN
		IF fbPump.bError THEN
			bError := TRUE;
			stError.ErrorId := fbPump.nErrorId;
			nStateAction := 99;
		ELSE
			nStateAction := 80;				
		END_IF
		fbPump(bExecute:= FALSE, DilSendCmd:= fbSendCmd, pDilRef:= pDiluterRef1);
	END_IF
END_IF

//Abbrechen
IF nStateAction = 70 THEN
	IF fbPump.bBusy THEN
		fbPump(bExecute:= FALSE, DilSendCmd:= fbSendCmd, pDilRef:= pDiluterRef1);
	ELSE
		nStateAction := 71;
	END_IF
END_IF

IF nStateAction = 71 THEN
	fbStop(bExecute:= TRUE, DilSendCmd:= fbSendCmd, pDilRef1 := pDiluterRef1);
	IF NOT fbStop.bBusy THEN
		IF fbStop.bError THEN
			nStateAction := 99;
			stError.ErrorId := fbStop.nErrorId;
		ELSE
			nStateAction := nStateNext;
		END_IF
		fbStop(bExecute:= FALSE, DilSendCmd:= fbSendCmd);
	END_IF	
END_IF
//Ende Abbrechen

//Errorhandling
IF nStateAction = 99 THEN
	fbPump(bExecute:= FALSE, DilSendCmd:= fbSendCmd, pDilRef:= pDiluterRef1);
	stError.Cmd := E_Action.ACTION_DilPump;
	stError.POUAction := E_POUACT.POUACT_A_Pump;
	fbErrorList.M_Add(stError);
END_IF
END_ACTION

METHOD FB_init : BOOL
VAR_INPUT
	bInitRetains : BOOL; // if TRUE, the retain variables are initialized (warm start / cold start)
	bInCopyCode : BOOL;  // if TRUE, the instance afterwards gets moved into the copy code (online change)
END_VAR
eObjectType := E_ObjectType.OBJECTTYPE_Diluter3Inputs;
eObjectGroup := E_ObjectGroup.OBJECTGROUP_Device;
eValveType := E_DilValveType.VALVETYPE_4Distribution;
END_METHOD

METHOD M_CheckBottles : ERRORID
VAR_INPUT
	nInputNr : USINT;
END_VAR
IF nInputNr >= 1 AND nInputNr <= 3 THEN
	IF NOT aSensSysLiquidBottle[aLiquidBottle[nInputNr]] THEN
		M_CheckBottles := E_ErrorIdCmd.ERRORID_LiquidBottleEmpty;
		RETURN;
	END_IF
END_IF
END_METHOD

METHOD M_ExeAction : ERRORID
VAR_INPUT
	refActionData	: REFERENCE TO ST_ActionData;
END_VAR

VAR
	i : USINT;
END_VAR
//Diluter kann keine Actions parallel ausführen
//Die einzige Action ist Stop
IF eCurrentState = E_MachineState.MACHINESTATE_Idle THEN
	CASE refActionData.eAction OF
		E_Action.ACTION_DilPump: //Diluter Pumpen
			IF NOT bIsInit THEN
				M_ExeAction := E_ErrorIdDiluter.ERRORID_NotIniialized;
				RETURN;
			END_IF
			//Param1 = Quantity in 10tel µl
			//Param2 = Mode (Saugen oder Drücken) //Hier wird nur Drücken implementiert!
			//Param3 = Flow Pumpen in 10tel µl/sec
			//Param4 = Flow Nachladen in 10tel µl/sec
			//Param5 = Ventilstellung Pump
			//Param6 = Ventilstellung Nachladen
			//Param7 = Ctrl (verschiedene Steuer-Bis (z.B. MoveBottom before Pump o.ä.)
			
			//Valve-Position Pumpen ist immer der Output wenn nicht anders angegeben.
			IF refActionData.aParams[5] = 0 THEN
				nValvePosPump := nValvePosOutput;
			ELSE
				nValvePosPump := DINT_TO_SINT(refActionData.aParams[5]);
			END_IF
			
			//Valve-Position Reload ermitteln
			IF refActionData.aParams[6] = 0 THEN
				//Dieser Fall sollte einen Fehler werfen, da keine eindeutige Zuordnung möglich ist.
				M_ExeAction := E_ErrorIdDiluter.ERRORID_InvalidValveParam;
			ELSE
				nValvePosReload := DINT_TO_SINT(refActionData.aParams[6]);
				IF nValvePosReload < 1 OR nValvePosReload > 4 THEN
					M_ExeAction := E_ErrorIdDiluter.ERRORID_InvalidValveParam;
					RETURN;
				END_IF
			END_IF
			
			nCurrentBottleNr := 0;
			ePumpMode := DINT_TO_USINT(refActionData.aParams[1]);
			//Überwachung der Bottles erfolgt nur im Pumpmode "Press", da Bottles Vorratsflaschen
			IF ePumpMode = E_DilPumpMode.MODE_Press THEN
				FOR i:= 1 TO 3 BY 1 DO
					IF aValvePosInput[i] = nValvePosReload THEN
						nCurrentBottleNr := i;
						EXIT;
					END_IF
				END_FOR
				
				M_ExeAction := M_CheckBottles(nCurrentBottleNr);
				IF M_ExeAction > 0 THEN
					RETURN;
				END_IF
			END_IF
			
			//Umrechnung von 10tel µl in Mircosteps
			nTotalSteps := F_DilQuantityToMicroSteps(refActionData.aParams[2],nSyringeSize);
			
			//Umrechnung 10tel µl/s in Halbsteps/s
			nSpeedPump := F_DilFlowToSpeed(refActionData.aParams[3], nSyringeSize);
	
			M_ExeAction := M_CheckSpeed(nSpeedPump);
			IF M_ExeAction > 0 THEN
				RETURN;
			END_IF
			
			IF refActionData.aParams[4] = 0 THEN
				//Umrechnung 10tel µl/s in Halbsteps/s
				nSpeedReload := F_DilFlowToSpeed(nConfigReloadSpeed, nSyringeSize);
			ELSE
				//Umrechnung 10tel µl/s in Halbsteps/s
				nSpeedReload := F_DilFlowToSpeed(refActionData.aParams[4], nSyringeSize);
			END_IF
			M_ExeAction := M_CheckSpeed(nSpeedReload);
			IF M_ExeAction > 0 THEN
				RETURN;
			END_IF			
			bPump := TRUE;
			
		E_Action.ACTION_DilTransfer:
			//Diese Action ist für diesen Dilutertyp nicht implementiert
				M_ExeAction := E_ErrorIdCmd.ERRORID_InvalidActionDiluterType;
				RETURN;
		E_Action.ACTION_DilPrepare:
			IF NOT bIsInit THEN
				M_ExeAction := E_ErrorIdDiluter.ERRORID_NotIniialized;
				RETURN;
			END_IF

			ePrepareMode := DINT_TO_USINT(refActionData.aParams[1]);
			nInput  := DINT_TO_USINT(refActionData.aParams[3]);
			IF nInput < 1 OR nInput > 3 THEN
				M_ExeAction := E_ErrorIdCmd.ERRORID_ActionLocked;
				RETURN;
			END_IF
			
			//Bottles OK?
			M_ExeAction := M_CheckBottles(nInput);
			IF M_ExeAction > 0 THEN
				RETURN;
			END_IF
			
			fbMoveToPos.nValvePos := aValvePosInput[nInput];
			
			//Umrechnung von 10tel µl in Mircosteps
			nTotalSteps := F_DilQuantityToMicroSteps(refActionData.aParams[2],nSyringeSize);
			nTotalSteps := MIN(24000,nTotalSteps);	//Es kann für max einen Hub reloaded werden
			nSpeedReload := F_DilFlowToSpeed(nConfigReloadSpeed, nSyringeSize);
			
			bPrepare := TRUE;
		ELSE
			M_ExeAction := SUPER^.M_ExeAction(refActionData);
			RETURN;
	END_CASE
	bBusy := TRUE;
	eCurrentAction := refActionData.eAction;
	eCurrentState := E_MachineState.MACHINESTATE_Active;
ELSIF (eCurrentState = E_MachineState.MACHINESTATE_Active) AND (refActionData.eAction = E_Action.ACTION_Stop) THEN
	M_Stop();
ELSE
	M_ExeAction := E_ErrorIdCmd.ERRORID_InvalidState;
	RETURN;
END_IF
END_METHOD

METHOD M_GetAllProps : ERRORID
VAR_INPUT
	refCmdData : REFERENCE TO  ST_CmdData;
END_VAR
//Specialproperties lesen
refCmdData.aHeader[0] := nObjectID;
refCmdData.aHeader[1] := eObjectType;
refCmdData.aHeader[2]:= nNotifyId;

refCmdData.n32Data[1] := nParentSlotNr;
refCmdData.n32Data[2] := nChannel;		//Diluter-Kanal
refCmdData.n32Data[3] := nSyringeSize;	//Spritzengröße (für beide Dilutoren)
refCmdData.n32Data[4] := nConfigReloadSpeed;
refCmdData.n32Data[5] := aLiquidBottle[1];
refCmdData.n32Data[6] := aLiquidBottle[2];
refCmdData.n32Data[7] := aLiquidBottle[3];
refCmdData.n32Data[8] := aValvePosInput[1];
refCmdData.n32Data[9] := aValvePosInput[2];
refCmdData.n32Data[10] := aValvePosInput[3];
refCmdData.n32Data[11] := nValvePosOutput;
END_METHOD

METHOD M_GetValvePosInput : SINT
VAR_INPUT
	nInputNr : USINT;
END_VAR
IF nInputNr >= 1 AND nInputNr <= 3 THEN
	M_GetValvePosInput := aValvePosInput[nInputNr];
END_IF
END_METHOD

METHOD M_SetAllProps : ERRORID
VAR_INPUT
	refCmdData : REFERENCE TO  ST_CmdData;
END_VAR
nNoOfProps := 12;

nParentSlotNr := DINT_TO_UINT(refCmdData.n32Data[1]);

//Diluterkanal checken
//Channel muss zwischen 1 und 7 liegen
IF  NOT((refCmdData.n32Data[2] > 0) AND (refCmdData.n32Data[2] <= cNoOfDiluters)) THEN
	M_SetAllProps := E_ErrorIdObjMgmt.ERRORID_InvalidDiluterChannel;
	RETURN;
ELSE
	nChannel := DINT_TO_USINT(refCmdData.n32Data[2]);
	pDiluterRef1 := ADR(aFbDiluterRef[nChannel]);
END_IF

//Spritzengröße
IF NOT (refCmdData.n32Data[3] = 50 OR 
		refCmdData.n32Data[3] = 100 OR 
		refCmdData.n32Data[3] = 250 OR 
		refCmdData.n32Data[3] = 500 OR 
		refCmdData.n32Data[3] = 1000 OR
		refCmdData.n32Data[3] = 2500 OR
		refCmdData.n32Data[3] = 5000) THEN
		M_SetAllProps := E_ErrorIdObjMgmt.ERRORID_InvalidSyringeSize;
ELSE
	nSyringeSize := refCmdData.n32Data[3];
END_IF

//ReloadSpeed
nConfigReloadSpeed := refCmdData.n32Data[4];

//Liquidbottle 1
IF refCmdData.n32Data[5] >= 0 AND refCmdData.n32Data[5] <= cNoOfLiquidBottles THEN
	aLiquidBottle[1] := DINT_TO_USINT(refCmdData.n32Data[5]);
ELSE
	M_SetAllProps := E_ErrorIdObjMgmt.ERRORID_InvalidLiquidbottle;
	RETURN;
END_IF

//Liquidbottle 2
IF refCmdData.n32Data[6] >= 0 AND refCmdData.n32Data[6] <= cNoOfLiquidBottles THEN
	aLiquidBottle[2] := DINT_TO_USINT(refCmdData.n32Data[6]);
ELSE
	M_SetAllProps := E_ErrorIdObjMgmt.ERRORID_InvalidLiquidbottle;
	RETURN;
END_IF

//Liquidbottle 3
IF refCmdData.n32Data[7] >= 0 AND refCmdData.n32Data[7] <= cNoOfLiquidBottles THEN
	aLiquidBottle[3] := DINT_TO_USINT(refCmdData.n32Data[7]);
ELSE
	M_SetAllProps := E_ErrorIdObjMgmt.ERRORID_InvalidLiquidbottle;
	RETURN;
END_IF

//Achtung, ValvePos muss einen Wert von 1 bis 4 annehmen, denn dieser Diluter ist fix mit einem 4Way-Valve ausgestattet.
aValvePosInput[1] := DINT_TO_SINT(refCmdData.n32Data[8]);
aValvePosInput[2] := DINT_TO_SINT(refCmdData.n32Data[9]);
aValvePosInput[3] := DINT_TO_SINT(refCmdData.n32Data[10]);
nValvePosOutput := DINT_TO_SINT(refCmdData.n32Data[11]);
END_METHOD

END_FUNCTION_BLOCK

// ---- Hardware/MultiZ/FB_MultiZTipEjector.TcPOU
FUNCTION_BLOCK FB_MultiZTipEjector
VAR_INPUT
	pfbZAxisRef	: POINTER TO FB_ZAxisRef;
	bExecute 	: BOOL;	
END_VAR
VAR_OUTPUT
	bBusy : BOOL;
	bError : BOOL;
	nErrorId : ERRORID;	
END_VAR
VAR
	nState : USINT;
	tmrDelay : TON;
END_VAR

IF bExecute THEN
	bBusy := TRUE;
	IF pfbZAxisRef^.stInput.nError > 0 THEN
		pfbZAxisRef^.stStatus.bError := TRUE;
		bBusy := FALSE;
		bError := TRUE;
		nErrorId := F_MultiZError_TO_ErrorId(pfbZAxisRef^.stInput.nError);
		RETURN;
	END_IF
	
	CASE nState OF
		0:	pfbZAxisRef^.stOutput.nToolCtrl := 1;
			tmrDelay(IN:= TRUE, PT:=T#500MS);
			nState := 1;

		1:	tmrDelay();
			IF tmrDelay.Q THEN
				tmrDelay(IN:= FALSE);
				nState := 2;
			END_IF
			
		2:	IF NOT pfbZAxisRef^.stInput.nToolState.0 THEN
				pfbZAxisRef^.stOutput.nToolCtrl := 0;
				nState := 80;
				bBusy := FALSE;			
			END_IF
 	END_CASE
ELSE
	tmrDelay(IN:= FALSE);
	bBusy := FALSE;
	bError := FALSE;
	nErrorId := 0;
	nState := 0;
END_IF

END_FUNCTION_BLOCK

// ---- Objects/Targets/Passive/FB_Rack.TcPOU
FUNCTION_BLOCK FB_Rack EXTENDS FB_SlotTarget
VAR_INPUT
END_VAR
VAR_OUTPUT
END_VAR
VAR
END_VAR

METHOD M_GetAbsPos : ST_3DPoint
VAR_INPUT
	pChildPos	: POINTER TO ST_3DPoint;
	eTargetRef 	: E_TargetRef;
	nParam1		: UINT;
 	nParam2		: UINT;
	nParam3		: USINT;
	nParam4		: USINT;
	nZLevel		: USINT;
END_VAR
VAR_OUTPUT
	nErrorId 	: ERRORID;
	lrAngle		: LREAL;
END_VAR
VAR
	stLocPosLB : ST_3DPoint;
	pSlot : POINTER TO FB_PieceSlot;
END_VAR
IF eTargetRef = E_TargetRef.TARGETREF_Slot THEN
	//Slotnummer checken
	pSlot := super^.M_GetSlot(nParam1);
	IF pSlot > 0 THEN
		stLocPosLB := P_stRelPosLB;	//hier wird auch berücksichtigt, wenn das Rack an einem Slot hängt
		//Slot belegt?
		IF pSlot^.P_pPiece > 0 THEN
			stLocPosLB := F_Add3DPoints(stLocPosLB, pSlot^.P_pPiece^.M_GetRelPosTopCenter());
		ELSE
			stLocPosLB := F_Add3DPoints(stLocPosLB, pSlot^.P_stRelPos);
		END_IF
		
		M_GetAbsPos := pParentTarget^.M_GetAbsPos(pChildPos := ADR(stLocPosLB), eTargetRef:= E_TargetRef.TARGETREF_LeftBottom,
														nParam1:= 0,
														nParam2:= 0, nParam3:= 0, nParam4:= 0, nZLevel:= 0,
														lrAngle => lrAngle, nErrorId=> nErrorId);		
	ELSE
		nErrorId := E_ErrorIdCmd.ERRORID_InvalidTargetSlot;
	END_IF
	
ELSE
	M_GetAbsPos := SUPER^.M_GetAbsPos(pChildPos := pChildPos, eTargetRef:= eTargetRef,
													nParam1:= nParam1,
													nParam2:= nParam2, nParam3:= nParam3, nParam4:=0, nZLevel:= nZLevel,
													lrAngle => lrAngle, nErrorId=> nErrorId);	
END_IF
END_METHOD

METHOD M_GetNextFreeSlot : POINTER TO FB_SLOT
VAR_INPUT
	stRange : ST_Rectangle;
END_VAR
VAR
	pSlot 	: POINTER TO FB_PieceSlot;
END_VAR
fbSlotList.M_SetCurrentToHead();
REPEAT
	pSlot := fbSlotList.M_GetNext();
	IF pSlot > 0 THEN
		IF F_PointInnerRect(stPoint:= pSlot^.P_stAbsPos, stRectangle:= stRange) THEN
			IF pSlot^.P_pPiece = 0 THEN
				M_GetNextFreeSlot := pSlot;
				RETURN;
			END_IF			
		END_IF
	END_IF
UNTIL (pSlot = 0)
END_REPEAT
END_METHOD

METHOD M_GetNextFreshPieceSlot : POINTER TO FB_PieceSlot
VAR_INPUT
	stRange : ST_Rectangle;
END_VAR

VAR
	pSlot 	: POINTER TO FB_PieceSlot;
	pUsingPiece : POINTER TO FB_UsingPiece;
END_VAR
fbSlotList.M_SetCurrentToHead();
REPEAT
	pSlot := fbSlotList.M_GetNext();
	IF pSlot > 0 THEN
		IF F_PointInnerRect(stPoint:= pSlot^.P_stAbsPos, stRectangle:= stRange) THEN
			IF pSlot^.P_pPiece > 0 THEN
				IF pSlot^.P_pPiece^.bUsingPiece THEN
					pUsingPiece := pSlot^.P_pPiece;
					IF NOT pUsingPiece^.P_bUsed THEN
						M_GetNextFreshPieceSlot := pSlot;
						RETURN;
					END_IF
				ELSE
					M_GetNextFreshPieceSlot := pSlot;
				END_IF
			END_IF
		END_IF
	END_IF
UNTIL (pSlot = 0)
END_REPEAT
END_METHOD

END_FUNCTION_BLOCK

// ---- Objects/F_PointInnerRect.TcPOU
FUNCTION F_PointInnerRect : BOOL
VAR_INPUT
	stPoint		: ST_3DPoint;
	stRectangle : ST_Rectangle;
END_VAR
VAR
END_VAR

F_PointInnerRect := (stPoint.X >= stRectAngle.X1) AND
					(stPoint.X <= stRectAngle.X2) AND
					(stPoint.Y >= stRectAngle.Y1) AND
					(stPoint.Y <= stRectAngle.Y2);

END_FUNCTION

// ---- Objects/Pieces/FB_UsingPiece.TcPOU
FUNCTION_BLOCK FB_UsingPiece EXTENDS FB_PieceBase
VAR_INPUT
END_VAR
VAR_OUTPUT
END_VAR
VAR
	bUsed 	: BOOL;	
END_VAR

METHOD M_GetAllProps : ERRORID
VAR_INPUT
	refCmdData : REFERENCE TO  ST_CmdData;
END_VAR
SUPER^.M_GetAllProps(refCmdData);
nCurrentPropIndex := nCurrentPropIndex + 1;
refCmdData.n32Data[nCurrentPropIndex] := BOOL_TO_DINT(bUsed);
END_METHOD

METHOD M_SetSingleProp : ERRORID
VAR_INPUT
	refCmdData : REFERENCE TO  ST_CmdData;
END_VAR
IF refCmdData.aHeader[1] = nSpecPropIndex THEN
	bUsed := DINT_TO_BOOL(refCmdData.n32Data[0]);
ELSE
	M_SetSingleProp := SUPER^.M_SetSingleProp(refCmdData);
END_IF
END_METHOD

{attribute 'object_name' := 'M_SetAllProps'}
METHOD M_SetAllProps : ERRORID
VAR_INPUT
	refCmdData	: REFERENCE TO ST_CmdData;
END_VAR
M_SetAllProps := SUPER^.M_SetAllProps(refCmdData);

IF M_SetAllProps > 0 THEN
	RETURN;
END_IF
nCurrentPropIndex := nCurrentPropIndex + 1;
nSpecPropIndex := nCurrentPropIndex;

bUsed := DINT_TO_BOOL(refCmdData.n32Data[nCurrentPropIndex]);

nNoOfProps := nCurrentPropIndex + 1;
END_METHOD

PROPERTY P_bUsed : BOOL
GET
P_bUsed := bUsed;
END_GET
SET
bUsed := P_bUsed;
END_SET
END_PROPERTY

END_FUNCTION_BLOCK

// ---- Objects/Tools/FB_TwinPiezoHolder.TcPOU
FUNCTION_BLOCK FB_TwinPiezoHolder EXTENDS FB_GCodeTool
VAR_INPUT
END_VAR
VAR_OUTPUT
END_VAR
VAR
	//SpecProperties
	stPipIntxnPos			: ST_3DPoint;	//Relative Position des Schnittpunktes der eingeschwenkten Pipetten
	stPipIntxnOffset		: ST_3DPoint;	//Offset  des Schnittpunktes der eingeschwenkten Pipetten (z.B. durch Teachen)
	
	//****************************************Aktionvariablen****************************************************
	
	//Action: "InitTool"
	bInitTool			: BOOL;
	bInitSpecFlag		: BOOL := TRUE;
	nStateA_InitTool	: USINT;
	
	//Action: "Swivel"
	bSwivel				: BOOL;
	nStateA_Swivel		: USINT;
	eSwivelCtrl			: E_SwivelCtrl;
	
	//Action: "Aspirate"
	bAspirate			: BOOL;
	nStateA_Aspirate	: USINT;
	nQuantity			: DINT;
	nFlow				: DINT;
	
	//Action: "Dispense"
	bDispense			: BOOL;
	nStateA_Dispense	: USINT;
	
	//Action: "DispensePiezo"
	bDispensePiezo			: BOOL;
	nStateA_DispensePiezo	: USINT;
	nDrops1					: UINT;
	nDrops2					: UINT;
	bDispensePiezoStart		: BOOL;
	bStroboskopeOn			: BOOL;
	bSetDropsFlag			: BOOL := TRUE;	
	nTestResult				: UDINT;	//wird beim PiezoTest durch InteractResponse Arg1 geschrieben bzw. bei Start des Tests zurückgesetzt
	
	//Action: "MoveDilValve"
	bDilMoveValve			: BOOL;
	nStateA_DilMoveValve	: USINT;
	
	
	timeout				: TON;

	pPiezoRefMaster			: POINTER TO FB_PiezoRef;
	pPiezoRefSlave			: POINTER TO FB_PiezoRef;
	pPiezoPipFirst			: POINTER TO FB_PiezoPip;
	pPiezoPipSecond			: POINTER TO FB_PiezoPip;
	
	//Status
	eCurSwivelState			: E_SwivelState;
	
END_VAR

VAR CONSTANT
	cNumberOfSlots : UINT := 2;
END_VAR

IF eCurrentState = E_MachineState.MACHINESTATE_Active THEN
	IF bInitTool THEN
		A_InitTool();
		IF nStateA_InitTool >= 80 THEN
			IF nStateA_InitTool >= 99 THEN
				bError := TRUE;
			END_IF
			bInitTool := FALSE;
			nStateA_InitTool := 0;
			M_RemoveListEntry(nSearchValue:= E_Action.ACTION_Init);
		END_IF
	END_IF

	IF bAspirate THEN
		A_Aspirate();
		IF nStateA_Aspirate >= 80 THEN
			IF nStateA_Aspirate >= 99 THEN
				bError := TRUE;	
			END_IF
			bAspirate := FALSE;
			nStateA_Aspirate := 0;
			M_RemoveListEntry(nSearchValue:= E_Action.ACTION_Aspirate);
		END_IF
	END_IF

	IF bDispense THEN
		A_Dispense();
		IF nStateA_Dispense >= 80 THEN
			IF nStateA_Dispense >= 99 THEN
				bError := TRUE;	
			END_IF
			bDispense := FALSE;
			nStateA_Dispense := 0;
			M_RemoveListEntry(nSearchValue:= E_Action.ACTION_Dispense);
		END_IF
	END_IF
	
	IF bDispensePiezo THEN
		A_DispensePiezo();
		IF nStateA_DispensePiezo >= 80 THEN
			IF nStateA_DispensePiezo >= 99 THEN
				bError := TRUE;	
			END_IF
			bDispensePiezo := FALSE;
			nStateA_DispensePiezo := 0;
			M_RemoveListEntry(nSearchValue:= ACTION_DispenseDrops);
		END_IF
	END_IF
	
	IF bDilMoveValve THEN
		A_DilMoveValve();
		IF nStateA_DilMoveValve >= 80 THEN
			IF nStateA_DilMoveValve >= 99 THEN
				bError := TRUE;			
			END_IF
			bDilMoveValve := FALSE;
			nStateA_DilMoveValve := 0;
			M_RemoveListEntry(nSearchValue:= E_Action.ACTION_DilMoveValve);
		END_IF
	END_IF	

	IF bSwivel THEN
		A_Swivel();
		IF nStateA_Swivel >= 80 THEN
			IF nStateA_Swivel >= 99 THEN
				bError := TRUE;
			END_IF
			bSwivel := FALSE;
			nStateA_Swivel := 0;
			M_RemoveListEntry(nSearchValue:= E_Action.ACTION_Swivel);
		END_IF		
	END_IF
END_IF

SUPER^();	//FB_MzTool aufrufen

//Prozessdaten aktualisieren
stProcessData.n32Data[7] := eCurSwivelState;
stProcessData.n32Data[8] := BOOL_TO_DINT(bDispensePiezo);
aObjProcData[nNotifyId] := stProcessData;

ACTION A_Aspirate:
IF pPiezoPipSecond > 0 THEN
	IF pPiezoPipSecond^.P_pDiluter^.P_bError THEN
		stError.ErrorId := pPiezoPipSecond^.P_pDiluter^.P_nErrorId;
		stError.POUState := nStateA_Aspirate;
		nStateA_Aspirate := 99;		
	END_IF
END_IF

IF nStateA_Aspirate <> 99 THEN
	IF pPiezoPipFirst > 0 THEN
		IF pPiezoPipFirst^.P_pDiluter^.P_bError THEN
			stError.ErrorId := pPiezoPipFirst^.P_pDiluter^.P_nErrorId;
			stError.POUState := nStateA_Aspirate;
			nStateA_Aspirate := 99;		
		END_IF		
	END_IF
END_IF 

CASE nStateA_Aspirate OF
	0:	MEMSET(ADR(stActionData),0,SIZEOF(stActionData));
		stActionData.eAction := E_Action.ACTION_DilPump;
		stActionData.aParams[1] := E_DilPumpMode.MODE_Suck;
		stActionData.aParams[2] := nQuantity; 
		stActionData.aParams[3] := nFlow;
		//stActionDataSpec.aParams[4] := 0; //ReloadSpeed wird von DilConfig übernommen
		//stActionDataSpec.aParams[5] := 1; //Valve-Position für Pump
		//stActionDataSpec.aParams[6] := 2; //Valve-Position für Reload
		nStateA_Aspirate := 1;
		IF pPiezoPipSecond > 0 THEN
			stError.ErrorId := pPiezoPipSecond^.P_pDiluter^.M_ExeAction(stActionData);
		END_IF
		IF stError.ErrorId > 0 THEN
			nStateA_Aspirate := 99;
		ELSIF pPiezoPipFirst > 0 THEN
			stError.ErrorId := pPiezoPipFirst^.P_pDiluter^.M_ExeAction(stActionData);
			IF stError.ErrorId > 0 THEN
				nStateA_Aspirate := 99;
			END_IF
		END_IF
		
	1:	//Warten bis Aspiration fertig
		nStateA_Aspirate := 80;
		IF pPiezoPipSecond > 0 THEN
			IF pPiezoPipSecond^.P_pDiluter^.M_GetActionBusy(E_Action.ACTION_DilPump) THEN
				nStateA_Aspirate := 1;
			END_IF
		END_IF
		IF pPiezoPipFirst > 0 THEN
			IF pPiezoPipFirst^.P_pDiluter^.M_GetActionBusy(E_Action.ACTION_DilPump) THEN
				nStateA_Aspirate := 1;
			END_IF
		END_IF
		
	70:	//Abbrechen
		IF pPiezoPipSecond > 0 THEN
			pPiezoPipSecond^.P_pDiluter^.M_CancelAction(ACTION_DilPump);
		END_IF
		IF pPiezoPipFirst > 0 THEN
			pPiezoPipFirst^.P_pDiluter^.M_CancelAction(ACTION_DilPump);
		END_IF
		nStateA_Aspirate := 1;
END_CASE

//Errorhandling
IF nStateA_Aspirate = 99 THEN
	stError.Cmd := E_Action.ACTION_Aspirate;
	stError.POU := E_POU.POU_FB_PiezoPip;
	stError.POUAction := E_POUACT.POUACT_A_Aspirate;
	fbErrorList.M_Add(stError);
END_IF
END_ACTION

ACTION A_DilMoveValve:
stError.POUState := nStateA_DilMoveValve;

IF pPiezoPipFirst > 0 THEN
	IF pPiezoPipFirst^.P_bError THEN
		stError.ErrorId := 	pPiezoPipFirst^.P_nErrorId;
		nStateA_DilMoveValve := 99;
	END_IF
END_IF

IF pPiezoPipSecond > 0 THEN
	IF pPiezoPipSecond^.P_bError THEN
		stError.ErrorId := 	pPiezoPipSecond^.P_nErrorId;
		nStateA_DilMoveValve := 99;
	END_IF
END_IF

IF nStateA_DilMoveValve = 0 THEN
	nStateA_DilMoveValve := 80;
	IF pPiezoPipFirst > 0 THEN
		IF pPiezoPipFirst^.M_GetActionBusy(E_Action.ACTION_DilMoveValve) THEN
			nStateA_DilMoveValve := 0;
		END_IF
	END_IF

	IF pPiezoPipSecond > 0 THEN
		IF pPiezoPipSecond^.M_GetActionBusy(E_Action.ACTION_DilMoveValve) THEN
			nStateA_DilMoveValve := 0;
		END_IF
	END_IF
END_IF

//Errorhandling
IF nStateA_DilMoveValve = 99 THEN
	stError.Cmd := E_Action.ACTION_DilMoveValve;
	stError.POU := E_POU.POU_FB_PiezoPip;
	stError.POUAction := E_POUACT.POUACT_A_MoveValve;
	fbErrorList.M_Add(stError);
END_IF
END_ACTION

ACTION A_Dispense:
IF pPiezoPipSecond > 0 THEN
	IF pPiezoPipSecond^.P_pDiluter^.P_bError THEN
		stError.ErrorId := pPiezoPipSecond^.P_pDiluter^.P_nErrorId;
		stError.POUState := nStateA_Dispense;
		nStateA_Dispense := 99;		
	END_IF
END_IF

IF nStateA_Dispense <> 99 THEN
	IF pPiezoPipFirst > 0 THEN
		IF pPiezoPipFirst^.P_pDiluter^.P_bError THEN
			stError.ErrorId := pPiezoPipFirst^.P_pDiluter^.P_nErrorId;
			stError.POUState := nStateA_Dispense;
			nStateA_Dispense := 99;		
		END_IF		
	END_IF
END_IF 

CASE nStateA_Dispense OF
	0:	MEMSET(ADR(stActionData),0,SIZEOF(stActionData));
		stActionData.eAction := E_Action.ACTION_DilPump;
		stActionData.aParams[1] := E_DilPumpMode.MODE_Press;
		stActionData.aParams[2] := nQuantity; 
		stActionData.aParams[3] := nFlow;
		//stActionDataSpec.aParams[4] := 0; //ReloadSpeed wird von DilConfig übernommen
		//stActionDataSpec.aParams[5] := 1; //Valve-Position für Pump
		//stActionDataSpec.aParams[6] := 2; //Valve-Position für Reload
		nStateA_Dispense := 1;
		IF pPiezoPipSecond > 0 THEN
			stError.ErrorId := pPiezoPipSecond^.P_pDiluter^.M_ExeAction(stActionData);
		END_IF
		IF stError.ErrorId > 0 THEN
			nStateA_Dispense := 99;
		ELSIF pPiezoPipFirst > 0 THEN
			stError.ErrorId := pPiezoPipFirst^.P_pDiluter^.M_ExeAction(stActionData);
			IF stError.ErrorId > 0 THEN
				nStateA_Dispense := 99;
			END_IF
		END_IF
		
	1:	//Warten bis Dispensen fertig
		nStateA_Dispense := 80;
		IF pPiezoPipSecond > 0 THEN
			IF pPiezoPipSecond^.P_pDiluter^.M_GetActionBusy(E_Action.ACTION_DilPump) THEN
				nStateA_Dispense := 1;
			END_IF
		END_IF
		IF pPiezoPipFirst > 0 THEN
			IF pPiezoPipFirst^.P_pDiluter^.M_GetActionBusy(E_Action.ACTION_DilPump) THEN
				nStateA_Dispense := 1;
			END_IF
		END_IF
		
	70:	//Abbrechen
		IF pPiezoPipSecond > 0 THEN
			pPiezoPipSecond^.P_pDiluter^.M_CancelAction(ACTION_DilPump);
		END_IF
		IF pPiezoPipFirst > 0 THEN
			pPiezoPipFirst^.P_pDiluter^.M_CancelAction(ACTION_DilPump);
		END_IF
		nStateA_Dispense := 71;
		
	71:	//Warten bis Dispensen fertig
		nStateA_Dispense := 80;
		IF pPiezoPipSecond > 0 THEN
			IF pPiezoPipSecond^.P_pDiluter^.M_GetActionBusy(E_Action.ACTION_DilPump) THEN
				nStateA_Dispense := 71;
			END_IF
		END_IF
		IF pPiezoPipFirst > 0 THEN
			IF pPiezoPipFirst^.P_pDiluter^.M_GetActionBusy(E_Action.ACTION_DilPump) THEN
				nStateA_Dispense := 71;
			END_IF
		END_IF
END_CASE

//Errorhandling
IF nStateA_Dispense = 99 THEN
	stError.Cmd := E_Action.ACTION_Dispense;
	stError.POU := E_POU.POU_FB_PiezoPip;
	stError.POUAction := E_POUACT.POUACT_A_Dispense;
	fbErrorList.M_Add(stError);
END_IF
END_ACTION

ACTION A_DispensePiezo:
IF nStateA_DispensePiezo = 0 THEN
	MEMSET(ADR(stActionData),0,SIZEOF(stActionData));
	stActionData.eAction := E_Action.ACTION_DilMoveValve;
	stActionData.aParams[1] := 3; //Bypass-Stellung

	nStateA_DispensePiezo := 2;
	//Falls die Diluter noch nicht in Bypass stehen, diese erst in Bypass stellen
	//gestellt werden und somit die Pipetten nicht zeitgleich gestartet werden
	IF pPiezoPipFirst^.P_pDiluter^.P_nCurValvePos <> 3 THEN
		nStateA_DispensePiezo := 1;
		stError.ErrorId := pPiezoPipFirst^.P_pDiluter^.M_ExeAction(stActionData);
	END_IF
	
	IF stError.ErrorId > 0 THEN
		nStateA_DispensePiezo := 99;
	ELSE
		IF pPiezoPipSecond^.P_pDiluter^.P_nCurValvePos <> 3 THEN
			nStateA_DispensePiezo := 1;
			stError.ErrorId := pPiezoPipSecond^.P_pDiluter^.M_ExeAction(stActionData);
		END_IF
		IF stError.ErrorId > 0 THEN
			nStateA_DispensePiezo := 99;
		END_IF
	END_IF

ELSIF nStateA_DispensePiezo = 1 THEN	//Warten bis beide Diluter gestellt
	nStateA_DispensePiezo := 2;
	IF pPiezoPipSecond^.P_pDiluter^.M_GetActionBusy(E_Action.ACTION_DilMoveValve) THEN
		nStateA_DispensePiezo := 1;
	ELSE
		IF pPiezoPipSecond^.P_pDiluter^.P_bError THEN
			stError.ErrorId := pPiezoPipSecond^.P_pDiluter^.P_nErrorId;
			nStateA_DispensePiezo := 99;
		END_IF
	END_IF
	
	IF nStateA_DispensePiezo = 2 THEN
		IF pPiezoPipFirst^.P_pDiluter^.M_GetActionBusy(E_Action.ACTION_DilMoveValve) THEN
			nStateA_DispensePiezo := 1;
		ELSE
			IF pPiezoPipFirst^.P_pDiluter^.P_bError THEN
				stError.ErrorId := pPiezoPipFirst^.P_pDiluter^.P_nErrorId;
				nStateA_DispensePiezo := 99;
			END_IF
		END_IF		
	END_IF
END_IF

IF nStateA_DispensePiezo = 2 THEN	//Dispensen beide Pipetten starten
	nStateA_DispensePiezo := 3;
	pPiezoRefMaster^.P_bSynchronize := TRUE;
   	pPiezoRefSlave^.P_bSynchronize := TRUE;
	MEMSET(ADR(stActionData),0,SIZEOF(stActionData));
	stActionData.eAction := E_Action.ACTION_DispenseDrops;
	stActionData.aParams[1] := nDrops1;
	stActionData.aParams[2] := 1; //Start
	stError.ErrorId := pPiezoPipFirst^.M_ExeAction(stActionData);
	IF stError.ErrorId > 0 THEN
		nStateA_DispensePiezo := 99;
	ELSE
		stActionData.aParams[1] := nDrops2;
		stActionData.aParams[3] := BOOL_TO_DINT(bStroboskopeOn);
		stError.ErrorId := pPiezoPipSecond^.M_ExeAction(stActionData);
		IF stError.ErrorId > 0 THEN
			 pPiezoPipFirst^.M_CancelAction(E_Action.ACTION_DispenseDrops);
			nStateA_DispensePiezo := 99;
		END_IF
	END_IF
ELSIF nStateA_DispensePiezo = 3 THEN //Warten bis Dispensen fertig
	nStateA_DispensePiezo := 80;
	IF pPiezoPipFirst^.M_GetActionBusy(E_Action.ACTION_DispenseDrops) OR pPiezoPipSecond^.M_GetActionBusy(E_Action.ACTION_DispenseDrops) THEN
		nStateA_DispensePiezo := 3;
	ELSE
		IF pPiezoPipFirst^.P_bError THEN
			stError.ErrorId := pPiezoPipFirst^.P_nErrorId;
			nStateA_DispensePiezo := 99;
		END_IF
	END_IF
	
	IF nStateA_DispensePiezo = 80 THEN
		IF pPiezoPipSecond^.M_GetActionBusy(E_Action.ACTION_DispenseDrops) THEN
			nStateA_DispensePiezo := 3;
		ELSE
			IF pPiezoPipSecond^.P_bError THEN
				stError.ErrorId := pPiezoPipSecond^.P_nErrorId;
				nStateA_DispensePiezo := 99;
			END_IF
		END_IF
	END_IF
ELSIF nStateA_DispensePiezo = 70 THEN
	 pPiezoPipFirst^.M_CancelAction(E_Action.ACTION_DispenseDrops);
	 pPiezoPipSecond^.M_CancelAction(E_Action.ACTION_DispenseDrops);
	 nStateA_DispensePiezo := 80;
END_IF

//Errorhandling
IF nStateA_DispensePiezo = 99 THEN
	stError.Cmd := E_Action.ACTION_DispenseDrops;
	stError.POU := E_POU.POU_FB_PiezoPip;
	stError.POUAction := E_POUACT.POUACT_A_DispensePiezo;
	fbErrorList.M_Add(stError);
END_IF
END_ACTION

ACTION A_InitTool:
IF nStateA_InitTool = 0 THEN
	IF NOT bInitAxis THEN //Warten bis InitBase fertig
			bInitToolOk := FALSE;
			IF bError THEN
				nStateA_InitTool := 0;
				bInitTool := FALSE;
				M_RemoveListEntry(nSearchValue:= E_Action.ACTION_Init);
				RETURN;
			END_IF
			pZAxisRef^.stOutput.nToolCtrl.3 := TRUE; //Dispensermode "Piezo" (notwendig zum Schwenken)
			pZAxisRef^.stOutput.nToolCtrl.6 := TRUE; //Einschwenken
			timeout(IN:= TRUE, PT:= T#10S);
			eCurSwivelState := E_SwivelState.UNDEFINED;
			nStateA_InitTool := 1;
		END_IF
ELSIF nStateA_InitTool < 5	THEN
	nStateA_InitTool := nStateA_InitTool + 1;
ELSIF nStateA_InitTool = 5	THEN
	//Warten bis eingeschwenkt
	timeout();
	IF timeout.Q THEN
		timeout(IN:= FALSE);
		stError.ErrorId := E_ErrorIdMultiZ.ERRORID_TimeoutSwivel;
		nStateA_InitTool := 99;
	END_IF
	IF pZAxisRef^.stInput.nToolState.4 THEN
		timeout(IN:= FALSE);
		timeout(IN:= TRUE, PT:= T#10S);
		pZAxisRef^.stOutput.nToolCtrl.6 := FALSE; //Ausschwenken
		nStateA_InitTool := nStateA_InitTool + 1;
	END_IF
ELSIF nStateA_InitTool < 10 THEN
	nStateA_InitTool := nStateA_InitTool + 1;
ELSIF nStateA_InitTool = 10	THEN
	//Warten bis ausgeschwenkt
	timeout();
	IF timeout.Q THEN
		timeout(IN:= FALSE);
		stError.ErrorId := E_ErrorIdMultiZ.ERRORID_TimeoutSwivel;
		nStateA_InitTool := 99;
	END_IF
	IF NOT pZAxisRef^.stInput.nToolState.4 THEN
		timeout(IN:= FALSE);
		bInitToolOk := TRUE;
		eCurSwivelState := E_SwivelState.Original;
		nStateA_InitTool := 80;
	END_IF
ELSIF nStateA_InitTool = 70	THEN
	nStateA_InitTool := 80;
END_IF

//Errorhandling
IF nStateA_InitTool = 99 THEN
	stError.POU := E_POU.POU_FB_TwinPiezoHolder;
	stError.Cmd := E_Action.ACTION_Init;
	stError.POUAction := E_POUACT.POUACT_A_InitSpec;
	fbErrorList.M_Add(stError);
END_IF
END_ACTION

ACTION A_Reset:
//Ist noch eine Aktion aktiv?
IF nStateA_ResetSpec = 0 THEN 
	IF bAspirate THEN
		bAspirate := FALSE;
		nStateA_Aspirate := 0;
	END_IF

	IF bDispense THEN
		bDispense := FALSE;
		nStateA_Dispense := 0;
	END_IF

	IF bDispensePiezo THEN
		bDispensePiezo := FALSE;
		nStateA_DispensePiezo := 0;
	END_IF	
	
	IF bDilMoveValve THEN
		bDilMoveValve := FALSE;
		nStateA_DilMoveValve := 0;
	END_IF	
	
	nStateA_ResetSpec := 80;
END_IF

SUPER^.A_Reset();
END_ACTION

ACTION A_Stop:
IF nStateA_Stop = 0 THEN
	IF bInitTool AND nStateA_InitTool < 70 THEN
		nStateA_InitTool := 70;
	END_IF
	
	IF bAspirate AND nStateA_Aspirate < 70 THEN
		nStateA_Aspirate := 70;
	END_IF

	IF bDispense AND nStateA_Dispense < 70 THEN
		nStateA_Dispense := 70;
	END_IF

	IF bDispensePiezo AND nStateA_DispensePiezo < 70 THEN
		nStateA_DispensePiezo := 70;
	END_IF
	
	IF bSwivel AND nStateA_Swivel < 70 THEN
		nStateA_Swivel := 70;
	END_IF	

	nStateA_Stop := 1;
END_IF

SUPER^.A_Stop();
END_ACTION

ACTION A_Swivel:
//Schwenken wird nur in FreePos durchgeführt
IF nStateA_Swivel = 0 THEN
	IF P_bCollFree THEN
		nStateA_Swivel := 2;
	ELSE
		MEMSET(ADR(stActionData),0,SIZEOF(stActionData));
		stActionData.eAction := E_Action.ACTION_MoveZ;
		stActionData.aParams[1] := E_MoveMode.MODE_Free;
		stActionData.aParams[3] := -1; //MaxSpeed Z
		stError.ErrorId := M_ExeAction(stActionData);
		IF stError.ErrorId > 0 THEN	//Error
			nStateA_Swivel := 99;
		ELSE
			nStateA_Swivel := 1;
		END_IF
	END_IF
ELSIF nStateA_Swivel = 1 THEN //MoveZ-Free ready?
	IF NOT M_GetActionBusy(E_Action.ACTION_MoveZ) THEN
		nStateA_Swivel := 2;
	END_IF
END_IF

IF nStateA_Swivel = 2 THEN
		//State im ToolCtrl setzen
		pZAxisRef^.stOutput.nToolCtrl.6 := (eSwivelCtrl = E_SwivelCtrl.Swiveled);
		timeout(IN:= TRUE, PT:= T#10S);
		nStateA_Swivel := 3;
ELSIF nStateA_Swivel = 3 THEN
		eCurSwivelState := E_SwivelState.UNDEFINED;
		nStateA_Swivel := 4;
ELSIF nStateA_Swivel = 4 THEN
	//Warten bis ToolState entsprechend
	timeout();
	IF timeout.Q THEN
		timeout(IN:= FALSE);
		stError.ErrorId := E_ErrorIdMultiZ.ERRORID_TimeoutSwivel;
		nStateA_Swivel := 99;
	END_IF
	IF pZAxisRef^.stInput.nToolState.4 = pZAxisRef^.stOutput.nToolCtrl.6 THEN
		timeout(IN:= FALSE);
		IF eSwivelCtrl = E_SwivelCtrl.Swiveled THEN
			eCurSwivelState := E_SwivelState.Swiveled;
		ELSE
			eCurSwivelState := E_SwivelState.Original;
		END_IF
		nStateA_Swivel := 80;
	END_IF
END_IF

IF nStateA_Swivel = 70 THEN	//Abbrechen
	timeout(IN:= FALSE);
	nStateA_Swivel := 80;
END_IF

//Errorhandling
IF nStateA_InitTool = 99 THEN
	stError.POU := E_POU.POU_FB_TwinPiezoHolder;
	stError.Cmd := E_Action.ACTION_Swivel;
	stError.POUAction := E_POUACT.POUACT_A_Swivel;
	fbErrorList.M_Add(stError);
END_IF
END_ACTION

METHOD FB_init : BOOL
VAR_INPUT
	bInitRetains : BOOL; // if TRUE, the retain variables are initialized (warm start / cold start)
	bInCopyCode : BOOL;  // if TRUE, the instance afterwards gets moved into the copy code (online change)
END_VAR
eObjectType := E_ObjectType.OBJECTTYPE_TwinPiezoHolder;
eObjectGroup := E_ObjectGroup.OBJECTGROUP_MzTool OR E_ObjectGroup.OBJECTGROUP_Device;
END_METHOD

METHOD M_AddChild : ERRORID
VAR_INPUT
	pObject : POINTER TO FB_Object;
	nSlotNr	: UINT;
	nIndex 	: INT;
END_VAR
//Kann folgende Objekt-Typen aufnehmen
//Piezo, Solenoid
IF pObject > 0 THEN
	IF pObject^.P_eObjectType = E_ObjectType.OBJECTTYPE_PiezoPip OR
		pObject^.P_eObjectType = E_ObjectType.OBJECTTYPE_DummyTool OR
		pObject^.P_eObjectType = E_ObjectType.OBJECTTYPE_SolenoidPip THEN
		M_AddChild := SUPER^.M_AddChild(pObject,nSlotNr,nIndex);
	ELSE
		M_AddChild := E_ErrorIdObjMgmt.ERRORID_InvalidParentObject;
	END_IF
ELSE
	M_AddChild := E_ErrorIdObjMgmt.ERRORID_InvalidParentObject;
END_IF
END_METHOD

METHOD M_CancelAction
VAR_INPUT
	eAction : E_Action;
END_VAR
CASE eAction OF
	E_Action.ACTION_Aspirate:
		IF bAspirate AND nStateA_Aspirate < 70 THEN
			nStateA_Aspirate := 70;
		END_IF
	E_Action.ACTION_Dispense:
		IF bDispense AND nStateA_Dispense < 70 THEN
			nStateA_Dispense := 70;
		END_IF
	E_Action.ACTION_DispenseDrops:
		IF bDispensePiezo AND nStateA_DispensePiezo < 70 THEN
			nStateA_DispensePiezo := 70;
		END_IF
ELSE
	SUPER^.M_CancelAction(eAction);
END_CASE
END_METHOD

METHOD M_CheckAction : ERRORID
VAR_INPUT
	refActionData 	: REFERENCE TO ST_ActionData;
	pCorrelObject	: POINTER TO FB_Object;
END_VAR

VAR
END_VAR
CASE refActionData.eAction OF
	E_Action.ACTION_Dispense, //BasicAction für ActionOnArray
	E_Action.ACTION_DispenseDrops, //BasicAction für ActionOnArray
	E_Action.ACTION_DispenseTest,
	E_Action.ACTION_MoveToTarget,
	E_Action.ACTION_WashTool, E_Action.ACTION_GetPipSample:
		IF pPiezoPipFirst = 0 OR pPiezoPipSecond = 0 THEN
			M_CheckAction := E_ErrorIdCmd.ERRORID_NotAllPipettesConfigured;
		END_IF	
ELSE
	M_CheckAction := SUPER^.M_CheckAction(refActionData, pCorrelObject);
END_CASE
END_METHOD

METHOD M_CheckProps : ERRORID
VAR_INPUT
END_VAR

VAR
	pSlot : POINTER TO FB_Slot;
	pPiezo : POINTER TO FB_PiezoPip;
END_VAR
M_CheckProps := SUPER^.M_CheckProps();
//TwinPiezoHolder wird nur MzBase-Firmware mit Toolerkennung unterstützt
IF NOT NOT pFbMultiZ^.P_bLegacy THEN
	M_CheckProps := E_ErrorIdObjMgmt.ERRORID_FirmwareVersionMzBase;
	RETURN;
END_IF
fbSlotList.M_SetCurrentToHead();
pPiezoPipSecond := 0;
pPiezoPipFirst := 0;
REPEAT
	pSlot := fbSlotList.M_GetNext();
	IF pSlot > 0 THEN
		IF pSlot^.P_pChild > 0 THEN
			pPiezo := pSlot^.P_pChild;
			IF pPiezo^.P_pPiezoRef = pPiezoRefMaster THEN
				pPiezoPipSecond := pPiezo;
			ELSIF pPiezo^.P_pPiezoRef = pPiezoRefSlave THEN
				pPiezoPipFirst := pPiezo;
			END_IF
		END_IF
	END_IF
UNTIL (pSlot = 0)
END_REPEAT
END_METHOD

METHOD M_ExeAction : ERRORID
VAR_INPUT
	refActionData : REFERENCE TO ST_ActionData;	
END_VAR
IF NOT (eCurrentState = E_MachineState.MACHINESTATE_Idle OR
	eCurrentState = E_MachineState.MACHINESTATE_Active OR
	eCurrentState = E_MachineState.MACHINESTATE_Ready) THEN
	M_ExeAction := E_ErrorIdCmd.ERRORID_InvalidState;
	RETURN;
END_IF

CASE refActionData.eAction OF
	E_Action.ACTION_Init:
		IF NOT bInitAxis AND NOT bInitTool THEN
			bInitAxis := TRUE;
			bInitTool := TRUE;
			fbList.A_AddHeadValue(hList := hList, putValue := E_Action.ACTION_Init);	//InitAxis
			fbList.A_AddHeadValue(hList := hList, putValue := E_Action.ACTION_Init);	//InitTool
		ELSE
			RETURN;
		END_IF
		
	E_Action.ACTION_Aspirate:
		IF NOT bAspirate THEN
			IF (pPiezoPipFirst = 0) OR (pPiezoPipSecond = 0) THEN
				M_ExeAction := E_ErrorIdCmd.ERRORID_NotAllPipettesConfigured;
				RETURN;
			END_IF
			M_ExeAction := pPiezoPipFirst^.M_CheckBottles();
			IF M_ExeAction > 0 THEN
				RETURN;
			END_IF
			M_ExeAction := pPiezoPipSecond^.M_CheckBottles();
			IF M_ExeAction > 0 THEN
				RETURN;
			END_IF
			nQuantity := refActionData.aParams[1];
			nFlow := refActionData.aParams[2];
			fbList.A_AddHeadValue(hList:= hList, putValue:= E_Action.ACTION_Aspirate);
			bAspirate := TRUE;
		END_IF

	E_Action.ACTION_Dispense:
		IF NOT bDispense THEN
			IF (pPiezoPipFirst = 0) OR (pPiezoPipSecond = 0) THEN
				M_ExeAction := E_ErrorIdCmd.ERRORID_NotAllPipettesConfigured;
				RETURN;
			END_IF
			M_ExeAction := pPiezoPipFirst^.M_CheckBottles();
			IF M_ExeAction > 0 THEN
				RETURN;
			END_IF
			M_ExeAction := pPiezoPipSecond^.M_CheckBottles();
 			IF M_ExeAction > 0 THEN
				RETURN;
			END_IF
			nQuantity := refActionData.aParams[1];
			nFlow := refActionData.aParams[2];
			fbList.A_AddHeadValue(hList:= hList, putValue:= E_Action.ACTION_Dispense);
			bDispense := TRUE;
		END_IF
		
	E_Action.ACTION_DispenseDrops:
		IF (pPiezoPipSecond = 0) OR (pPiezoPipFirst = 0) THEN
			M_ExeAction := E_ErrorIdCmd.ERRORID_NotAllPipettesConfigured;
			RETURN;
		END_IF
 
		bDispensePiezoStart := DINT_TO_BOOL(refActionData.aParams[2]);
		
		IF (NOT bDispensePiezo) AND bDispensePiezoStart THEN
			nDrops1 := DINT_TO_UINT(refActionData.aParams[1]);
			bStroboskopeOn := DINT_TO_BOOL(refActionData.aParams[3]);
			nDrops2 := DINT_TO_UINT(refActionData.aParams[4]);
			fbList.A_AddHeadValue(hList:= hList, putValue := E_Action.ACTION_DispenseDrops);
			bDispensePiezo := TRUE;
		ELSIF bDispensePiezo AND (NOT bDispensePiezoStart) THEN
			pPiezoPipFirst^.M_CancelAction(E_Action.ACTION_DispenseDrops);
			pPiezoPipSecond^.M_CancelAction(E_Action.ACTION_DispenseDrops);
		ELSE
			RETURN;
		END_IF
		
	E_Action.ACTION_DilMoveValve:
		//Darf nur ausgeführt werden, wenn kein Dispensen aktiv ist
		IF NOT (bAspirate OR bDispense OR bDispensePiezo OR bDilMoveValve) THEN
			IF pPiezoPipFirst > 0 THEN
				M_ExeAction := pPiezoPipFirst^.M_ExeAction(refActionData);
			END_IF
			IF M_ExeAction > 0 THEN
				RETURN;
			ELSE
				IF pPiezoPipSecond > 0 THEN
					M_ExeAction := pPiezoPipSecond^.M_ExeAction(refActionData);
				END_IF
				IF M_ExeAction > 0 THEN
					RETURN;
				END_IF
			END_IF
			fbList.A_AddHeadValue(hList := hList, putValue := E_Action.ACTION_DilMoveValve);
			bDilMoveValve := TRUE;
		END_IF		
		
	E_Action.ACTION_Swivel:
		IF NOT bSwivel THEN
			bSwivel := TRUE;
			eSwivelCtrl := DINT_TO_USINT(refActionData.aParams[1]);
			fbList.A_AddHeadValue(hList := hList, putValue := E_Action.ACTION_Swivel);
		END_IF
	ELSE
		M_ExeAction := SUPER^.M_ExeAction(refActionData);
		RETURN;
END_CASE

bBusy := TRUE;
eCurrentState := E_MachineState.MACHINESTATE_Active;
END_METHOD

METHOD M_GetAllProps : ERRORID
VAR_INPUT
	refCmdData : REFERENCE TO  ST_CmdData;
END_VAR
//BaseProperties lesen
SUPER^.M_GetAllProps(refCmdData);
//BaseProperties lesen
nCurrentPropIndex := nCurrentPropIndex + 1;
refCmdData.n32Data[nCurrentPropIndex] := REAL_TO_DINT(stPipIntxnPos.X);
nCurrentPropIndex := nCurrentPropIndex + 1;
refCmdData.n32Data[nCurrentPropIndex] := REAL_TO_DINT(stPipIntxnPos.Y);
nCurrentPropIndex := nCurrentPropIndex + 1;
refCmdData.n32Data[nCurrentPropIndex] := REAL_TO_DINT(stPipIntxnPos.Z);
nCurrentPropIndex := nCurrentPropIndex + 1;
refCmdData.n32Data[nCurrentPropIndex] := REAL_TO_DINT(stPipIntxnOffset.X);
nCurrentPropIndex := nCurrentPropIndex + 1;
refCmdData.n32Data[nCurrentPropIndex] := REAL_TO_DINT(stPipIntxnOffset.Y);
nCurrentPropIndex := nCurrentPropIndex + 1;
refCmdData.n32Data[nCurrentPropIndex] := REAL_TO_DINT(stPipIntxnOffset.Z);
END_METHOD

METHOD M_GetPiezoRef : POINTER TO FB_PiezoRef
VAR_INPUT
	pToolSlot	: POINTER TO FB_Slot;
END_VAR
//Vorderansicht TwinPiezoHolder:
//links(Slot2) Master, rechts(Slot1) Slave 
IF pToolSlot^.P_nNr = 1 THEN //Slave
	M_GetPiezoRef := pPiezoRefSlave;
ELSIF pToolSlot^.P_nNr = 2 THEN //Master
	M_GetPiezoRef := pPiezoRefMaster;
END_IF
END_METHOD

METHOD M_SetAllProps : ERRORID
VAR_INPUT
	refCmdData : REFERENCE TO  ST_CmdData;
END_VAR
M_SetAllProps := SUPER^.M_SetAllProps(refCmdData);

IF M_SetAllProps > 0 THEN
	RETURN;
END_IF

//Spezi-Paramter schreiben
nCurrentPropIndex := nCurrentPropIndex + 1;
nSpecPropIndex := nCurrentPropIndex;
stPipIntxnPos.X := DINT_TO_REAL(refCmdData.n32Data[nCurrentPropIndex]);
nCurrentPropIndex := nCurrentPropIndex + 1;
stPipIntxnPos.Y := DINT_TO_REAL(refCmdData.n32Data[nCurrentPropIndex]);
nCurrentPropIndex := nCurrentPropIndex + 1;
stPipIntxnPos.Z := DINT_TO_REAL(refCmdData.n32Data[nCurrentPropIndex]);
nCurrentPropIndex := nCurrentPropIndex + 1;
stPipIntxnOffset.X := DINT_TO_REAL(refCmdData.n32Data[nCurrentPropIndex]);
nCurrentPropIndex := nCurrentPropIndex + 1;
stPipIntxnOffset.Y := DINT_TO_REAL(refCmdData.n32Data[nCurrentPropIndex]);
nCurrentPropIndex := nCurrentPropIndex + 1;
stPipIntxnOffset.Z := DINT_TO_REAL(refCmdData.n32Data[nCurrentPropIndex]);

//Die PiezoRef Master entspricht immer dem Achsenkanal, auf dem der Holder montiert ist
//Die PiezoRef Slave ist immer Achsenkanal - 1, ausser der Holder ist auf Achse1 montiert.
//In diesem Fall ist PiezoRef Slave = 2
//Der Master beansprucht das Schwenken für sich

pZAxisRef^.eFixedToolType := E_MzToolType.TOOL_TYPE_PiezoMaster;
IF pParentSlot^.P_nNr = 1 THEN
	pFbMultiZ^.aFbZAxisRef[2].eFixedToolType := E_MzToolType.TOOL_TYPE_PiezoSlave;
	pPiezoRefMaster := ADR(pFbMultiZ^.aFbPiezoRef[1]);
	pPiezoRefSlave := ADR(pFbMultiZ^.aFbPiezoRef[2]);
ELSE
	pFbMultiZ^.aFbZAxisRef[pParentSlot^.P_nNr - 1].eFixedToolType := E_MzToolType.TOOL_TYPE_PiezoSlave;
	pPiezoRefMaster := ADR(pFbMultiZ^.aFbPiezoRef[pParentSlot^.P_nNr]);
	pPiezoRefSlave := ADR(pFbMultiZ^.aFbPiezoRef[pParentSlot^.P_nNr - 1]);
END_IF
nNoOfProps := nCurrentPropIndex + 1;
END_METHOD

METHOD M_SetPrintParams : ST_MethResult
VAR_INPUT
	eType 		: E_PrintParamType;
	nNumerator	: USINT;
	nValue		: DINT;
END_VAR
CASE eType OF
	E_PrintParamType.Frequency:
		IF nNumerator = 1 THEN
			IF pPiezoPipFirst > 0 THEN
				M_SetPrintParams.nErrorId := pPiezoPipFirst^.M_SetFrequency(nValue, TRUE);
			ELSE
				M_SetPrintParams.nErrorId := E_ErrorIdCmd.ERRORID_InvalidPrintParamNumerator;	
			END_IF
		ELSIF nNumerator = 2 THEN
			IF pPiezoPipSecond > 0 THEN
				M_SetPrintParams.nErrorId := pPiezoPipSecond^.M_SetFrequency(nValue, TRUE);
			ELSE
				M_SetPrintParams.nErrorId := E_ErrorIdCmd.ERRORID_InvalidPrintParamNumerator;	
			END_IF
		ELSE
			M_SetPrintParams.nErrorId := E_ErrorIdCmd.ERRORID_InvalidPrintParamNumerator;
		END_IF
	E_PrintParamType.Pulse:
		IF nNumerator = 1 THEN
			IF pPiezoPipFirst > 0 THEN
				M_SetPrintParams.nErrorId := pPiezoPipFirst^.M_SetPulse(nValue, TRUE);
			ELSE
				M_SetPrintParams.nErrorId := E_ErrorIdCmd.ERRORID_InvalidPrintParamNumerator;	
			END_IF
		ELSIF nNumerator = 2 THEN
			IF pPiezoPipSecond > 0 THEN
				M_SetPrintParams.nErrorId := pPiezoPipSecond^.M_SetPulse(nValue, TRUE);
			ELSE
				M_SetPrintParams.nErrorId := E_ErrorIdCmd.ERRORID_InvalidPrintParamNumerator;	
			END_IF
		ELSE
			M_SetPrintParams.nErrorId := E_ErrorIdCmd.ERRORID_InvalidPrintParamNumerator;
		END_IF
	E_PrintParamType.Voltage:
		IF nNumerator = 1 THEN
			IF pPiezoPipFirst > 0 THEN
				M_SetPrintParams.nErrorId := pPiezoPipFirst^.M_SetVoltage(nValue, TRUE);
			ELSE
				M_SetPrintParams.nErrorId := E_ErrorIdCmd.ERRORID_InvalidPrintParamNumerator;	
			END_IF
		ELSIF nNumerator = 2 THEN
			IF pPiezoPipSecond > 0 THEN
				M_SetPrintParams.nErrorId := pPiezoPipSecond^.M_SetVoltage(nValue, TRUE);
			ELSE
				M_SetPrintParams.nErrorId := E_ErrorIdCmd.ERRORID_InvalidPrintParamNumerator;	
			END_IF
		ELSE
			M_SetPrintParams.nErrorId := E_ErrorIdCmd.ERRORID_InvalidPrintParamNumerator;
		END_IF
ELSE
	M_SetPrintParams.nErrorId := E_ErrorIdCmd.ERRORID_InvalidPrintParamType;
END_CASE

IF M_SetPrintParams.nErrorId > 0 THEN
	M_SetPrintParams.bError := TRUE;
END_IF
END_METHOD

METHOD M_SetSingleProp : ERRORID
VAR_INPUT
	refCmdData : REFERENCE TO  ST_CmdData;
END_VAR
IF nSpecPropIndex = refCmdData.aHeader[1] THEN
	stPipIntxnPos.X := DINT_TO_REAL(refCmdData.n32Data[0]);
ELSIF (nSpecPropIndex + 1) = refCmdData.aHeader[1] THEN
	stPipIntxnPos.Y := DINT_TO_REAL(refCmdData.n32Data[0]);
ELSIF (nSpecPropIndex + 2) = refCmdData.aHeader[1] THEN
	stPipIntxnPos.Z := DINT_TO_REAL(refCmdData.n32Data[0]);
ELSIF (nSpecPropIndex + 3) = refCmdData.aHeader[1] THEN
	stPipIntxnOffset.X := DINT_TO_REAL(refCmdData.n32Data[0]);
ELSIF (nSpecPropIndex + 4) = refCmdData.aHeader[1] THEN
	stPipIntxnOffset.Y := DINT_TO_REAL(refCmdData.n32Data[0]);
ELSIF (nSpecPropIndex + 5) = refCmdData.aHeader[1] THEN
	stPipIntxnOffset.Z := DINT_TO_REAL(refCmdData.n32Data[0]);
ELSE
	M_SetSingleProp := SUPER^.M_SetSingleProp(refCmdData);	
END_IF
END_METHOD

METHOD M_StartUniDispense : ERRORID
VAR_INPUT
	nParam1 : DINT; //Drops Pipette 1
	nParam2 : DINT; //Drops Pipette 2
END_VAR

VAR_OUTPUT
	bIsContinous : BOOL;
END_VAR

VAR
	stActionData : ST_ActionData;
END_VAR
stActionData.eAction := E_Action.ACTION_DispenseDrops;
stActionData.aParams[1] := nParam1;
stActionData.aParams[4] := nParam2;
stActionData.aParams[2] := 1; //On

IF nParam1 = 0 OR nParam2 = 0 THEN //DauerDispensen
	bIsContinous := TRUE;
END_IF

M_StartUniDispense := M_ExeAction(stActionData);
END_METHOD

METHOD M_StopUniDispense : ERRORID
VAR_INPUT
END_VAR
M_CancelAction(E_Action.ACTION_DispenseDrops);
END_METHOD

PROPERTY P_bIsInit : BOOL
GET
P_bIsInit := bInitToolOk AND SUPER^.P_bIsInit;
END_GET
END_PROPERTY

PROPERTY P_eCurrentSwivelState : E_SwivelState
GET
P_eCurrentSwivelState := eCurSwivelState;
END_GET
END_PROPERTY

PROPERTY P_pPiezoPipFirst : POINTER TO FB_PiezoPip
GET
P_pPiezoPipFirst := pPiezoPipFirst;
END_GET
END_PROPERTY

PROPERTY P_pPiezoPipSecond : POINTER TO FB_PiezoPip
GET
P_pPiezoPipSecond := pPiezoPipSecond;
END_GET
END_PROPERTY

PROPERTY P_stAbsPosPhys : ST_3DPoint
GET
VAR
	stTemp	: ST_3DPoint;
	stDim	: ST_3DDimension;
END_VAR
//Die absolute Postion eines Tool in "Z" hat nicht den gleichen Bezug wie X und Y
//X und Y beziehen sich auf den Koordinatenursprung, wenn die Achsen theoretisch aus Antrieb (0;0) stehen
//Z bezieht sich auf die Sliderunterkante des Z-Antriebes verechnet mit AbsPos vom Head(Ergebnis ist in den meisten Fällen negativ)

stTemp := F_Add3DPoints(stRelPos,stOffset);
//AbsPos vom ParentSlot holen
IF pParentSlot > 0 THEN
	stTemp := F_Add3DPoints(stTemp,pParentSlot^.P_stAbsPos);
END_IF

stTemp := F_Add3DPoints(stTemp,stPipIntxnPos);
P_stAbsPosPhys := F_Add3DPoints(stTemp,stPipIntxnOffset);
END_GET
END_PROPERTY

END_FUNCTION_BLOCK

// ---- Objects/Tools/FB_PiezoPip.TcPOU
FUNCTION_BLOCK FB_PiezoPip EXTENDS FB_GCodeTool IMPLEMENTS I_UsingDryPad
VAR_INPUT
END_VAR
VAR_OUTPUT
END_VAR
VAR
	//Specproperties
	nDiluterObjId		: UINT;
	pDiluter			: POINTER TO FB_Diluter;
	
	
	nDrypadArea			: USINT;
	tDryTime			: TIME;
	pFbPiezoRef			: POINTER TO FB_PiezoRef;
	fbPiezoControl		: FB_PiezoControl;
	pFbHeaterRef		: POINTER TO FB_MZHeaterRef;
	
	//****************************************Aktionvariablen****************************************************
	
	stActionDataSpec	: ST_ActionData;
	
	//Action: "InitTool"
	bInitTool			: BOOL;
	nStateA_InitTool	: USINT;	
	
	//Action: "Heating"
	bHeating 			: BOOL;
	nStateA_Heating		: USINT;		//State von A_Heating()
	nTempSetpoint		: UINT;			//Solltemperatur
	bHeatingOn			: BOOL;			//Heizung "EIN"	
	fbHeaterCtrl		: FB_MzHeaterControl;
	
	//Action: "Aspirate"
	bAspirate			: BOOL;
	nStateA_Aspirate	: USINT;
	nQuantity			: DINT;
	nFlow				: DINT;
	
	//Action: "Dispense"
	bDispense			: BOOL;
	nStateA_Dispense	: USINT;
	bSkipValveMove		: BOOL;	//wird benötigt, wenn DispenseDrops und Dispense gleichzeitig ausgeführt werden sollen (WashTool)

	//Action: "DispensePiezo"
	bDispensePiezo			: BOOL;
	nStateA_DispensePiezo	: USINT;
	nDrops					: UINT;
	bDispensePiezoStart		: BOOL;
	bStroboskopeOn			: BOOL;
	bSetDropsFlag			: BOOL := TRUE;	
	nTestResult				: UDINT;	//wird beim PiezoTest durch InteractResponse Arg1 geschrieben bzw. bei Start des Tests zurückgesetzt
	
	//Action: "MoveDilValve"
	bDilMoveValve			: BOOL;
	nStateA_DilMoveValve	: USINT;
	
END_VAR

fbPiezoControl(pFbPiezoRef:= pFbPiezoRef);

IF eCurrentState = E_MachineState.MACHINESTATE_Active THEN
	
	IF bInitTool THEN
		A_InitTool();
		IF nStateA_InitTool >= 80 THEN
			IF nStateA_InitTool >= 99 THEN
				bError := TRUE;
			END_IF
			bInitTool := FALSE;
			nStateA_InitTool := 0;
			M_RemoveListEntry(nSearchValue:= E_Action.ACTION_Init);
		END_IF		
	END_IF
	
	IF bHeating THEN	//Heizen
		A_Heating();
		IF nStateA_Heating >= 80 THEN
			IF nStateA_Heating >= 99 THEN
				bError := TRUE;
			END_IF
			bHeating := FALSE;
			nStateA_Heating := 0;
			M_RemoveListEntry(nSearchValue:= E_Action.ACTION_Heating);
		END_IF
	END_IF	
	
	IF bAspirate THEN
		A_Aspirate();
		IF nStateA_Aspirate >= 80 THEN
			IF nStateA_Aspirate >= 99 THEN
				bError := TRUE;	
			END_IF
			bAspirate := FALSE;
			nStateA_Aspirate := 0;
			M_RemoveListEntry(nSearchValue:= E_Action.ACTION_Aspirate);
		END_IF
	END_IF

	IF bDispense THEN
		A_Dispense();
		IF nStateA_Dispense >= 80 THEN
			IF nStateA_Dispense >= 99 THEN
				bError := TRUE;	
			END_IF
			bDispense := FALSE;
			nStateA_Dispense := 0;
			M_RemoveListEntry(nSearchValue:= E_Action.ACTION_Dispense);
		END_IF
	END_IF
	
	IF bDispensePiezo THEN
		A_DispensePiezo();
		IF nStateA_DispensePiezo >= 80 THEN
			IF nStateA_DispensePiezo >= 99 THEN
				bError := TRUE;			
			END_IF
			bDispensePiezo := FALSE;
			nStateA_DispensePiezo := 0;
			M_RemoveListEntry(nSearchValue:= E_Action.ACTION_DispenseDrops);
		END_IF
	END_IF
	
	IF bDilMoveValve THEN
		A_DilMoveValve();
		IF nStateA_DilMoveValve >= 80 THEN
			IF nStateA_DilMoveValve >= 99 THEN
				bError := TRUE;			
			END_IF
			bDilMoveValve := FALSE;
			nStateA_DilMoveValve := 0;
			M_RemoveListEntry(nSearchValue:= E_Action.ACTION_DilMoveValve);
		END_IF
	END_IF
END_IF

SUPER^();	//FB_MzTool aufrufen

//Prozessdaten aktualisieren
IF pFbPiezoRef > 0 THEN
	stProcessData.n32Data[7] := UDINT_TO_DINT(nTestResult);
	stProcessData.n32Data[10] := BOOL_TO_DINT(pFbPiezoRef^.pToolState^.0);
END_IF

IF pFbHeaterRef > 0 THEN
	stProcessData.n32Data[8] := BOOL_TO_DINT(pFbHeaterRef^.bHeaterIsOn);
	stProcessData.n32Data[9] := pFbHeaterRef^.nTemp1Actual;
END_IF

aObjProcData[nNotifyId] := stProcessData;

ACTION A_Aspirate:
IF pDiluter^.P_bError THEN
	stError.ErrorId := pDiluter^.P_nErrorId;
	stError.POUState := nStateA_Aspirate;
	nStateA_Aspirate := 99;
END_IF

CASE nStateA_Aspirate OF
	0:	MEMSET(ADR(stActionDataSpec),0,SIZEOF(stActionDataSpec));
		stActionDataSpec.eAction := E_Action.ACTION_DilPump;
		stActionDataSpec.aParams[1] := E_DilPumpMode.MODE_Suck;
		stActionDataSpec.aParams[2] := nQuantity; 
		stActionDataSpec.aParams[3] := nFlow;
		//stActionDataSpec.aParams[4] := 0; //ReloadSpeed wird von DilConfig übernommen
		//stActionDataSpec.aParams[5] := 1; //Valve-Position für Pump
		//stActionDataSpec.aParams[6] := 2; //Valve-Position für Reload
		
		stError.ErrorId := pDiluter^.M_ExeAction(stActionDataSpec);
		IF stError.ErrorId > 0 THEN
			stError.POUState := nStateA_Aspirate;
			nStateA_Aspirate := 99;
		ELSE
			nStateA_Aspirate := 1;	
		END_IF
		
	1:	//Warten bis Aspiration fertig
		IF NOT pDiluter^.M_GetActionBusy(E_Action.ACTION_DilPump) THEN
			nStateA_Aspirate := 80;
		END_IF
		
	70:	//Abbrechen
		MEMSET(ADR(stActionDataSpec),0,SIZEOF(stActionDataSpec));
		stActionDataSpec.eAction := E_Action.ACTION_Stop;
		
		pDiluter^.M_ExeAction(stActionDataSpec);
		nStateA_Aspirate := 71;
		
	71:	//Abbrechen
		IF NOT pDiluter^.P_bBusy THEN
			nStateA_Aspirate := 80;
		END_IF
END_CASE

//Errorhandling
IF nStateA_Aspirate = 99 THEN
	stError.Cmd := E_Action.ACTION_Aspirate;
	stError.POU := E_POU.POU_FB_PiezoPip;
	stError.POUAction := E_POUACT.POUACT_A_Aspirate;
	fbErrorList.M_Add(stError);
END_IF
END_ACTION

ACTION A_DilMoveValve:
stError.POUState := nStateA_DilMoveValve;
IF pDiluter^.P_bError THEN
	stError.ErrorId := pDiluter^.P_nErrorId;
	nStateA_DilMoveValve := 99;
END_IF

IF nStateA_DilMoveValve = 0 THEN
	IF NOT pDiluter^.M_GetActionBusy(E_Action.ACTION_DilMoveValve) THEN
		nStateA_DilMoveValve := 80;
	END_IF
END_IF

//Errorhandling
IF nStateA_DilMoveValve = 99 THEN
	stError.Cmd := E_Action.ACTION_DilMoveValve;
	stError.POU := E_POU.POU_FB_PiezoPip;
	stError.POUAction := E_POUACT.POUACT_A_MoveValve;
	fbErrorList.M_Add(stError);
END_IF
END_ACTION

ACTION A_Dispense:
IF pDiluter^.P_bError THEN
	stError.ErrorId := pDiluter^.P_nErrorId;
	stError.POUState := nStateA_Dispense;
	nStateA_Dispense := 99;
END_IF

CASE nStateA_Dispense OF
	0:	MEMSET(ADR(stActionDataSpec),0,SIZEOF(stActionDataSpec));
		////stActionDataSpec.bIntern := TRUE;
		stActionDataSpec.eAction := E_Action.ACTION_DilPump;
		stActionDataSpec.aParams[1] := E_DilPumpMode.MODE_Press;
		stActionDataSpec.aParams[2] := nQuantity; 
		stActionDataSpec.aParams[3] := nFlow;
		//stActionDataSpec.aParams[4] := 0;	//ReloadSpeed von DilConfig nehmen
		//stActionDataSpec.aParams[5] := 1; //Valve-Position für Pump
		//stActionDataSpec.aParams[6] := 2; //Valve-Position für Reload
		IF nQuantity = 0 THEN
			stActionDataSpec.aParams[7] := 1; //Endless
		END_IF
		
		stError.ErrorId := pDiluter^.M_ExeAction(stActionDataSpec);
		IF stError.ErrorId > 0 THEN
			stError.POUState := nStateA_Dispense;
			nStateA_Dispense := 99;
		ELSE
			nStateA_Dispense := 1;	
		END_IF
		
	1:	//Warten bis Dispensen fertig
		IF NOT pDiluter^.M_GetActionBusy(E_Action.ACTION_DilPump) THEN
			nStateA_Dispense := 80;
		END_IF
		
	70:	//Abbrechen
		MEMSET(ADR(stActionDataSpec),0,SIZEOF(stActionDataSpec));
		////stActionDataSpec.bIntern := TRUE;
		stActionDataSpec.eAction := E_Action.ACTION_Stop;
		
		pDiluter^.M_ExeAction(stActionDataSpec);
		nStateA_Dispense := 71;
		
	71:	
		IF NOT pDiluter^.P_bBusy THEN
			nStateA_Dispense := 80;
		END_IF
		
END_CASE

//Errorhandling
IF nStateA_Dispense = 99 THEN
	stError.Cmd := E_Action.ACTION_Dispense;
	stError.POU := E_POU.POU_FB_PiezoPip;
	stError.POUAction := E_POUACT.POUACT_A_Dispense;
	fbErrorList.M_Add(stError);
END_IF
END_ACTION

ACTION A_DispensePiezo:
CASE nStateA_DispensePiezo OF
	0:	//Wenn Diluter nicht auf Bypass, dann auf Bypass stellen
		IF bSkipValveMove THEN
			nStateA_DispensePiezo := 1;
		ELSE
			IF pDiluter^.P_nCurValvePos <> 3 THEN
				MEMSET(ADR(stActionDataSpec),0,SIZEOF(stActionDataSpec));
				stActionDataSpec.eAction := E_Action.ACTION_DilMoveValve;
				stActionDataSpec.aParams[1] := 3;
				stError.ErrorId := pDiluter^.M_ExeAction(stActionDataSpec);
				IF stError.ErrorId > 0 THEN
					stError.POUState := nStateA_DispensePiezo;
					nStateA_DispensePiezo := 99;
				ELSE
					nStateA_DispensePiezo := 1;
				END_IF
			ELSE
				nStateA_DispensePiezo := 1;
			END_IF
		END_IF
	
	1:	//Warten, bis Diluter fertig und Drops übertragen
		IF pDiluter^.P_bError THEN
			stError.ErrorId := pDiluter^.P_nErrorId;	
			stError.POUState := nStateA_DispensePiezo;
			nStateA_DispensePiezo := 99;
		ELSE
			IF (NOT pDiluter^.M_GetActionBusy(E_Action.ACTION_DilMoveValve)) AND nDrops = fbPiezoControl.P_nDrops THEN
				fbPiezoControl.M_StartStop(bDispensePiezoStart); //Piezo starten
				nStateA_DispensePiezo := 2;
			END_IF
		END_IF
		
	2: 	//Warten bis Piezo fertig
		IF NOT fbPiezoControl.bBusy THEN
			nStateA_DispensePiezo := 80;	
		END_IF
		
		IF fbPiezoControl.bError THEN
			stError.ErrorId := fbPiezoControl.nErrorId;
			stError.POUState := nStateA_DispensePiezo;
			nStateA_DispensePiezo := 99;
		END_IF
		
	70:	//Abbrechen
		fbPiezoControl.M_StartStop(FALSE);
		nStateA_DispensePiezo := 80;		
 END_CASE

//Errorhandling
IF nStateA_DispensePiezo = 99 THEN
	stError.Cmd := E_Action.ACTION_DispenseDrops;
	stError.POU := E_POU.POU_FB_PiezoPip;
	stError.POUAction := E_POUACT.POUACT_A_DispensePiezo;
	fbErrorList.M_Add(stError);
END_IF
END_ACTION

ACTION A_Heating:
IF nStateA_Heating = 0 THEN
	fbHeaterCtrl(bExecute:= TRUE, nTempZone1:= nTempSetpoint, bHeatingOn:= bHeatingOn, pFbHeaterRef:= pFbHeaterRef);

	IF NOT fbHeaterCtrl.bBusy THEN
		IF fbHeaterCtrl.bError THEN
			stError.ErrorId := fbHeaterCtrl.nErrorId; 
			stError.POUState := nStateA_Heating;
			nStateA_Heating := 99;
		ELSE
			nStateA_Heating := 80;	
		END_IF
		fbHeaterCtrl(bExecute:= FALSE, pFbHeaterRef:= pFbHeaterRef);
	END_IF
ELSIF nStateA_Heating = 70 THEN
	fbHeaterCtrl(bExecute:= FALSE, pFbHeaterRef:= pFbHeaterRef);
	nStateA_Heating := 80;
END_IF

//Errorhandling
IF nStateA_Heating = 99 THEN
	stError.POU := E_POU.POU_FB_PiezoPip;
	stError.Cmd := E_Action.ACTION_Heating;
	stError.POUAction := E_POUACT.POUACT_A_Heating;
	fbErrorList.M_Add(stError);
END_IF
END_ACTION

ACTION A_InitTool:
IF nStateA_InitTool = 0 THEN
	pFbPiezoRef^.P_eDispenserMode := E_DispenserMode.MODE_Piezo;
	fbPiezoControl.M_Init();
	bInitToolOk := TRUE;
	nStateA_InitTool := 80;
END_IF
END_ACTION

ACTION A_Reset:
//Ist noch eine Aktion aktiv?
IF nStateA_ResetSpec = 0 THEN 
	IF bAspirate THEN
		bAspirate := FALSE;
		nStateA_Aspirate := 0;
	END_IF

	IF bDispense THEN
		bDispense := FALSE;
		nStateA_Dispense := 0;
	END_IF

	IF bDispensePiezo THEN
		bDispensePiezo := FALSE;
		nStateA_DispensePiezo := 0;
	END_IF	
	
	IF bHeating THEN
		bHeating := FALSE;
		nStateA_Heating := 0;
	END_IF	
	
	nStateA_ResetSpec := 80;
END_IF

SUPER^.A_Reset();
END_ACTION

ACTION A_Stop:
IF nStateA_Stop = 0 THEN

	IF bAspirate AND nStateA_Aspirate < 70 THEN
		nStateA_Aspirate := 70;
	END_IF

	IF bDispense AND nStateA_Dispense < 70 THEN
		nStateA_Dispense := 70;
	END_IF

	IF bDispensePiezo AND nStateA_DispensePiezo < 70 THEN
		nStateA_DispensePiezo := 70;
	END_IF
	
	IF bHeating AND nStateA_Heating < 70 THEN
		nStateA_Heating := 70;
	END_IF
	
	nStateA_Stop := 1;
END_IF

SUPER^.A_Stop();
END_ACTION

METHOD FB_init : BOOL
VAR_INPUT
	bInitRetains : BOOL; // if TRUE, the retain variables are initialized (warm start / cold start)
	bInCopyCode : BOOL;  // if TRUE, the instance afterwards gets moved into the copy code (online change)
END_VAR
eObjectType := E_ObjectType.OBJECTTYPE_PiezoPip;
eObjectGroup := E_ObjectGroup.OBJECTGROUP_MzTool OR E_ObjectGroup.OBJECTGROUP_Device;
END_METHOD

METHOD M_AddChild : ERRORID
VAR_INPUT
	pObject : POINTER TO FB_Object;
	nSlotNr	: UINT;
	nIndex 	: INT;
END_VAR
//Kann keine Objekte aufnehmen
M_AddChild := E_ErrorIdObjMgmt.ERRORID_ObjectCanNotTakeChilds;
END_METHOD

METHOD M_CancelAction
VAR_INPUT
	eAction : E_Action;
END_VAR
CASE eAction OF
	E_Action.ACTION_Aspirate:
		IF bAspirate AND nStateA_Aspirate < 70 THEN
			nStateA_Aspirate := 70;
		END_IF
	E_Action.ACTION_Dispense:
		IF bDispense AND nStateA_Dispense < 70 THEN
			nStateA_Dispense := 70;
		END_IF
	E_Action.ACTION_DispenseDrops:
		IF bDispensePiezo AND nStateA_DispensePiezo < 70 THEN
			nStateA_DispensePiezo := 70;
		END_IF
	E_Action.ACTION_Heating:
		IF bHeating AND nStateA_Heating < 70 THEN
			nStateA_Heating := 70;
		END_IF	
ELSE
	SUPER^.M_CancelAction(eAction);
END_CASE
END_METHOD

METHOD M_CheckAction : ERRORID
VAR_INPUT
	refActionData 	: REFERENCE TO ST_ActionData;
	pCorrelObject	: POINTER TO FB_Object;
END_VAR

VAR
	pTarget : POINTER TO FB_TargetBase;
	pRack	: POINTER TO FB_Rack;
	pSlot	: POINTER TO FB_PieceSlot;
END_VAR
CASE refActionData.eAction OF
	E_Action.ACTION_GetPipSample,
	E_Action.ACTION_Dispense, //BasicAction für ActionOnArray
	E_Action.ACTION_Aspirate, //BasicAction für ActionOnArray
	E_Action.ACTION_DispenseDrops, //BasicAction für ActionOnArray
	E_Action.ACTION_DispenseTest,
	E_Action.ACTION_MeasureTool,
	E_Action.ACTION_TeachTarget:
		RETURN;
	E_Action.ACTION_WashTool:
		//Washmode checken
		IF refActionData.aParams[2] = E_WashMode.MODE_WashInside THEN
			M_CheckAction := M_CheckBottles();
		ELSIF refActionData.aParams[2] = E_WashMode.MODE_WashOutside THEN
			;
		ELSIF refActionData.aParams[2] = E_WashMode.MODE_WashInOutside THEN
			M_CheckAction := M_CheckBottles();
		ELSE
			M_CheckAction := E_ErrorIdCmd.ERRORID_InvalidWashMode;	
		END_IF
	E_Action.ACTION_InsertTool:
		//PiezoPip darf nur in offene Vials eintauchen
		//-> Target muss also ein VialRack sein (Reaktor nicht möglich, da Pip nicht von der Tiefe hinein passt)
		pTarget := pCorrelObject;
		IF pTarget > 0 THEN
			IF (pTarget^.P_eObjectGroup AND E_ObjectGroup.OBJECTGROUP_Rack) = E_ObjectGroup.OBJECTGROUP_Rack THEN
				pRack := pTarget;
				pSlot := pRack^.M_GetSlot(DINT_TO_UINT(refActionData.aParams[2]));
				IF pSlot > 0 THEN
					IF pSlot^.P_pPiece = 0 THEN
						M_CheckAction := E_ErrorIdCmd.ERRORID_NoPieceInSlot;
						RETURN;
					ELSIF NOT (pSlot^.P_pPiece^.P_eObjectType = E_ObjectType.OBJECTTYPE_Vial OR pSlot^.P_pPiece^.P_eObjectType = E_ObjectType.OBJECTTYPE_FlipTube) THEN
						M_CheckAction := E_ErrorIdCmd.ERRORID_InvalidPieceType;
					END_IF
				ELSE
					M_CheckAction := E_ErrorIdCmd.ERRORID_InvalidTargetSlot;
					RETURN;
				END_IF	
			ELSE
				M_CheckAction := E_ErrorIdCmd.ERRORID_UnsuitableTarget;	
			END_IF
		ELSE
			M_CheckAction := E_ErrorIdCmd.ERRORID_UnsuitableTarget;	
		END_IF	
ELSE
	M_CheckAction := SUPER^.M_CheckAction(refActionData, pCorrelObject);
END_CASE
END_METHOD

METHOD M_CheckBottles : ERRORID
VAR_INPUT
END_VAR
IF pDiluter > 0 THEN
	M_CheckBottles := pDiluter^.M_CheckBottles(0);
END_IF
END_METHOD

